LIN {X 0,Y 412.001,Z 515.214,A -85,B 0,C 180,E1 20178.098,E2 20178.098} C_VEL
LIN {X 0,Y 410.849,Z 527.535,A -85,B 0,C 180,E1 20175.962,E2 20175.962} C_VEL
LIN {X 0,Y 409.965,Z 537.694,A -85,B 0,C 180,E1 20173.828,E2 20173.828} C_VEL
LIN {X 0,Y 409.279,Z 546.504,A -85,B 0,C 180,E1 20171.556,E2 20171.556} C_VEL
LIN {X 0,Y 408.795,Z 553.889,A -85,B 0,C 180,E1 20169.148,E2 20169.148} C_VEL
LIN {X 0,Y 408.509,Z 559.483,A -85,B 0,C 180,E1 20166.747,E2 20166.747} C_VEL
LIN {X 0,Y 408.352,Z 563.605,A -85,B 0,C 180,E1 20164.213,E2 20164.213} C_VEL
LIN {X 0,Y 408.3,Z 565.991,A -85,B 0,C 180,E1 20161.684,E2 20161.684} C_VEL
LIN {X 0,Y 408.33,Z 566.694,A -85,B 0,C 180,E1 20159.158,E2 20159.158} C_VEL
LIN {X 0,Y 408.415,Z 565.71,A -85,B 0,C 180,E1 20156.632,E2 20156.632} C_VEL
LIN {X 0,Y 408.601,Z 563.017,A -85,B 0,C 180,E1 20154.101,E2 20154.101} C_VEL
LIN {X 0,Y 408.959,Z 558.554,A -85,B 0,C 180,E1 20151.565,E2 20151.565} C_VEL
LIN {X 0,Y 409.485,Z 552.563,A -85,B 0,C 180,E1 20149.163,E2 20149.163} C_VEL
LIN {X 0,Y 410.267,Z 544.675,A -85,B 0,C 180,E1 20146.757,E2 20146.757} C_VEL
LIN {X 0,Y 411.283,Z 535.28,A -85,B 0,C 180,E1 20144.49,E2 20144.49} C_VEL
LIN {X 0,Y 412.49,Z 524.341,A -85,B 0,C 180,E1 20142.363,E2 20142.363} C_VEL
LIN {X 0,Y 413.923,Z 511.401,A -85,B 0,C 180,E1 20140.308,E2 20140.308} C_VEL
LIN {X 0,Y 415.368,Z 497.854,A -85,B 0,C 180,E1 20138.538,E2 20138.538} C_VEL
LIN {X 0,Y 416.946,Z 482.078,A -85,B 0,C 180,E1 20136.842,E2 20136.842} C_VEL
LIN {X 0,Y 418.392,Z 465.945,A -85,B 0,C 180,E1 20135.429,E2 20135.429} C_VEL
LIN {X 0,Y 419.811,Z 447.969,A -85,B 0,C 180,E1 20134.161,E2 20134.161} C_VEL
LIN {X 0,Y 420.947,Z 429.995,A -85,B 0,C 180,E1 20133.173,E2 20133.173} C_VEL
LIN {X 0,Y 421.921,Z 409.848,A -85,B 0,C 180,E1 20132.352,E2 20132.352} C_VEL
LIN {X 0,Y 422.702,Z 387.891,A -85,B 0,C 180,E1 20131.742,E2 20131.742} C_VEL
LIN {X 0,Y 426.509,Z 310.931,A -85,B 0,C 180,E1 20129.855,E2 20129.855} C_VEL
LIN {X 0,Y 432.615,Z 224.265,A -85,B 0,C 180,E1 20127.543,E2 20127.543} C_VEL
LIN {X 0,Y 433.99,Z 205.725,A -85,B 0,C 180,E1 20127.01,E2 20127.01} C_VEL
LIN {X 0,Y 433.256,Z 198.82,A -85,B 0,C 180,E1 20126.606,E2 20126.606} C_VEL
LIN {X 0,Y 435.606,Z 168.281,A -85,B 0,C 180,E1 20123.85,E2 20123.85} C_VEL
LIN {X 0,Y 433.108,Z 159.078,A -85,B 0,C 180,E1 20122.283,E2 20122.283} C_VEL
LIN {X 0,Y 431.039,Z 153.151,A -85,B 0,C 180,E1 20120.995,E2 20120.995} C_VEL
LIN {X 0,Y 428.796,Z 147.265,A -85,B 0,C 180,E1 20119.416,E2 20119.416} C_VEL
LIN {X 0,Y 427.075,Z 143.317,A -85,B 0,C 180,E1 20117.916,E2 20117.916} C_VEL
LIN {X 0,Y 425.454,Z 140.615,A -85,B 0,C 180,E1 20115.735,E2 20115.735} C_VEL
LIN {X 0,Y 425.373,Z 139.927,A -85,B 0,C 180,E1 20114.891,E2 20114.891} C_VEL
LIN {X 0,Y 423.798,Z 146.299,A -85,B 0,C 180,E1 20113.08,E2 20113.08} C_VEL
LIN {X 0,Y 423.759,Z 151.293,A -85,B 0,C 180,E1 20111.84,E2 20111.84} C_VEL
LIN {X 0,Y 429.231,Z 165.38,A -85,B 0,C 180,E1 20109.893,E2 20109.893} C_VEL
LIN {X 0,Y 433.001,Z 172.844,A -85,B 0,C 180,E1 20109.358,E2 20109.358} C_VEL
LIN {X 0,Y 435.532,Z 195.035,A -85,B 0,C 180,E1 20108.647,E2 20108.647} C_VEL
LIN {X 0,Y 429.296,Z 412.636,A -85,B 0,C 180,E1 20104.609,E2 20104.609} C_VEL
LIN {X 0,Y 428.191,Z 433.533,A -85,B 0,C 180,E1 20104.074,E2 20104.074} C_VEL
LIN {X 0,Y 426.623,Z 453.74,A -85,B 0,C 180,E1 20103.327,E2 20103.327} C_VEL
LIN {X 0,Y 424.705,Z 474.23,A -85,B 0,C 180,E1 20102.305,E2 20102.305} C_VEL
LIN {X 0,Y 422.546,Z 493.789,A -85,B 0,C 180,E1 20101.055,E2 20101.055} C_VEL
LIN {X 0,Y 420.285,Z 512.438,A -85,B 0,C 180,E1 20099.581,E2 20099.581} C_VEL
LIN {X 0,Y 418.096,Z 529.523,A -85,B 0,C 180,E1 20097.952,E2 20097.952} C_VEL
LIN {X 0,Y 415.867,Z 546.483,A -85,B 0,C 180,E1 20096.027,E2 20096.027} C_VEL
LIN {X 0,Y 413.81,Z 562.406,A -85,B 0,C 180,E1 20093.874,E2 20093.874} C_VEL
LIN {X 0,Y 412.081,Z 576.353,A -85,B 0,C 180,E1 20091.643,E2 20091.643} C_VEL
LIN {X 0,Y 410.629,Z 589.282,A -85,B 0,C 180,E1 20089.192,E2 20089.192} C_VEL
LIN {X 0,Y 409.52,Z 600.704,A -85,B 0,C 180,E1 20086.599,E2 20086.599} C_VEL
LIN {X 0,Y 408.748,Z 610.548,A -85,B 0,C 180,E1 20083.871,E2 20083.871} C_VEL
LIN {X 0,Y 408.316,Z 618.348,A -85,B 0,C 180,E1 20081.155,E2 20081.155} C_VEL
LIN {X 0,Y 408.116,Z 624.334,A -85,B 0,C 180,E1 20078.454,E2 20078.454} C_VEL
LIN {X 0,Y 408.063,Z 628.633,A -85,B 0,C 180,E1 20075.767,E2 20075.767} C_VEL
LIN {X 0,Y 408.071,Z 631.328,A -85,B 0,C 180,E1 20073.091,E2 20073.091} C_VEL
LIN {X 0,Y 408.085,Z 632.331,A -85,B 0,C 180,E1 20070.422,E2 20070.422} C_VEL
LIN {X 0,Y 408.075,Z 631.775,A -85,B 0,C 180,E1 20067.754,E2 20067.754} C_VEL
LIN {X 0,Y 408.06,Z 629.669,A -85,B 0,C 180,E1 20065.081,E2 20065.081} C_VEL
LIN {X 0,Y 408.086,Z 625.91,A -85,B 0,C 180,E1 20062.398,E2 20062.398} C_VEL
LIN {X 0,Y 408.22,Z 620.753,A -85,B 0,C 180,E1 20059.844,E2 20059.844} C_VEL
LIN {X 0,Y 408.554,Z 613.61,A -85,B 0,C 180,E1 20057.133,E2 20057.133} C_VEL
LIN {X 0,Y 409.151,Z 605.098,A -85,B 0,C 180,E1 20054.553,E2 20054.553} C_VEL
LIN {X 0,Y 410.081,Z 594.653,A -85,B 0,C 180,E1 20051.963,E2 20051.963} C_VEL
LIN {X 0,Y 411.428,Z 581.988,A -85,B 0,C 180,E1 20049.368,E2 20049.368} C_VEL
LIN {X 0,Y 413.037,Z 568.55,A -85,B 0,C 180,E1 20047.063,E2 20047.063} C_VEL
LIN {X 0,Y 414.922,Z 553.715,A -85,B 0,C 180,E1 20044.906,E2 20044.906} C_VEL
LIN {X 0,Y 417.057,Z 537.409,A -85,B 0,C 180,E1 20042.903,E2 20042.903} C_VEL
LIN {X 0,Y 419.4,Z 519.234,A -85,B 0,C 180,E1 20041.037,E2 20041.037} C_VEL
LIN {X 0,Y 421.766,Z 500.31,A -85,B 0,C 180,E1 20039.437,E2 20039.437} C_VEL
LIN {X 0,Y 423.939,Z 481.065,A -85,B 0,C 180,E1 20038.109,E2 20038.109} C_VEL
LIN {X 0,Y 425.899,Z 461.768,A -85,B 0,C 180,E1 20037.047,E2 20037.047} C_VEL
LIN {X 0,Y 427.63,Z 441.297,A -85,B 0,C 180,E1 20036.184,E2 20036.184} C_VEL
LIN {X 0,Y 429.023,Z 419.453,A -85,B 0,C 180,E1 20035.539,E2 20035.539} C_VEL
LIN {X 0,Y 434.819,Z 218.607,A -85,B 0,C 180,E1 20031.785,E2 20031.785} C_VEL
LIN {X 0,Y 435.397,Z 192.267,A -85,B 0,C 180,E1 20031.286,E2 20031.286} C_VEL
LIN {X 0,Y 432.688,Z 171.767,A -85,B 0,C 180,E1 20030.595,E2 20030.595} C_VEL
LIN {X 0,Y 428.726,Z 164.272,A -85,B 0,C 180,E1 20030.006,E2 20030.006} C_VEL
LIN {X 0,Y 421.635,Z 146.282,A -85,B 0,C 180,E1 20027.418,E2 20027.418} C_VEL
LIN {X 0,Y 414.514,Z 130.026,A -85,B 0,C 180,E1 20024.835,E2 20024.835} C_VEL
LIN {X 0,Y 410.976,Z 122.341,A -85,B 0,C 180,E1 20023.512,E2 20023.512} C_VEL
LIN {X 0,Y 409.495,Z 119.111,A -85,B 0,C 180,E1 20022.94,E2 20022.94} C_VEL
LIN {X 0,Y 409.394,Z 118.478,A -85,B 0,C 180,E1 20022.802,E2 20022.802} C_VEL
LIN {X 0,Y 409.381,Z 118.43,A -85,B 0,C 180,E1 20019.045,E2 20019.045} C_VEL
LIN {X 0,Y 409.389,Z 118.489,A -85,B 0,C 180,E1 20015.099,E2 20015.099} C_VEL
LIN {X 0,Y 409.387,Z 118.49,A -85,B 0,C 180,E1 20011.183,E2 20011.183} C_VEL
LIN {X 0,Y 409.385,Z 118.487,A -85,B 0,C 180,E1 20007.253,E2 20007.253} C_VEL
LIN {X 0,Y 409.384,Z 118.474,A -85,B 0,C 180,E1 20003.307,E2 20003.307} C_VEL
LIN {X 0,Y 409.383,Z 118.471,A -85,B 0,C 180,E1 19999.4,E2 19999.4} C_VEL
LIN {X 0,Y 409.382,Z 118.488,A -85,B 0,C 180,E1 19995.439,E2 19995.439} C_VEL
LIN {X 0,Y 409.383,Z 118.482,A -85,B 0,C 180,E1 19991.553,E2 19991.553} C_VEL
LIN {X 0,Y 409.384,Z 118.465,A -85,B 0,C 180,E1 19987.72,E2 19987.72} C_VEL
LIN {X 0,Y 409.395,Z 118.489,A -85,B 0,C 180,E1 19983.921,E2 19983.921} C_VEL
LIN {X 0,Y 409.405,Z 118.465,A -85,B 0,C 180,E1 19980.14,E2 19980.14} C_VEL
LIN {X 0,Y 409.416,Z 118.476,A -85,B 0,C 180,E1 19976.359,E2 19976.359} C_VEL
LIN {X 0,Y 409.427,Z 118.48,A -85,B 0,C 180,E1 19972.422,E2 19972.422} C_VEL
LIN {X 0,Y 409.416,Z 118.461,A -85,B 0,C 180,E1 19968.448,E2 19968.448} C_VEL
LIN {X 0,Y 409.426,Z 118.482,A -85,B 0,C 180,E1 19964.562,E2 19964.562} C_VEL
LIN {X 0,Y 409.417,Z 118.478,A -85,B 0,C 180,E1 19960.601,E2 19960.601} C_VEL
LIN {X 0,Y 409.417,Z 118.463,A -85,B 0,C 180,E1 19956.668,E2 19956.668} C_VEL
LIN {X 0,Y 409.417,Z 118.47,A -85,B 0,C 180,E1 19952.669,E2 19952.669} C_VEL
LIN {X 0,Y 409.419,Z 118.484,A -85,B 0,C 180,E1 19948.73,E2 19948.73} C_VEL
LIN {X 0,Y 409.409,Z 118.488,A -85,B 0,C 180,E1 19944.805,E2 19944.805} C_VEL
LIN {X 0,Y 409.423,Z 118.489,A -85,B 0,C 180,E1 19940.764,E2 19940.764} C_VEL
LIN {X 0,Y 409.407,Z 118.486,A -85,B 0,C 180,E1 19936.857,E2 19936.857} C_VEL
LIN {X 0,Y 409.429,Z 118.668,A -85,B 0,C 180,E1 19932.947,E2 19932.947} C_VEL
LIN {X 0,Y 416.973,Z 136.874,A -85,B 0,C 180,E1 19929.573,E2 19929.573} C_VEL
LIN {X 0,Y 423.523,Z 154.25,A -85,B 0,C 180,E1 19926.674,E2 19926.674} C_VEL
LIN {X 0,Y 428.061,Z 168.125,A -85,B 0,C 180,E1 19924.581,E2 19924.581} C_VEL
LIN {X 0,Y 427.595,Z 173.606,A -85,B 0,C 180,E1 19924.047,E2 19924.047} C_VEL
LIN {X 0,Y 433.281,Z 207.319,A -85,B 0,C 180,E1 19922.841,E2 19922.841} C_VEL
LIN {X 0,Y 429.712,Z 391.959,A -85,B 0,C 180,E1 19919.803,E2 19919.803} C_VEL
LIN {X 0,Y 428.766,Z 411.13,A -85,B 0,C 180,E1 19919.244,E2 19919.244} C_VEL
LIN {X 0,Y 427.491,Z 428.701,A -85,B 0,C 180,E1 19918.497,E2 19918.497} C_VEL
LIN {X 0,Y 425.737,Z 446.594,A -85,B 0,C 180,E1 19917.482,E2 19917.482} C_VEL
LIN {X 0,Y 424.972,Z 453.23,A -85,B 0,C 180,E1 19917.028,E2 19917.028} C_VEL
LIN {X 0,Y 423.297,Z 460.11,A -85,B 0,C 180,E1 19916.595,E2 19916.595} C_VEL
LIN {X 0,Y 416.045,Z 476.098,A -85,B 0,C 180,E1 19915.6,E2 19915.6} C_VEL
LIN {X 0,Y 413.969,Z 482.401,A -85,B 0,C 180,E1 19915.045,E2 19915.045} C_VEL
LIN {X 0,Y 413.808,Z 483.266,A -85,B 0,C 180,E1 19914.953,E2 19914.953} C_VEL
LIN {X 0,Y 411.333,Z 498.226,A -85,B 0,C 180,E1 19913.189,E2 19913.189} C_VEL
LIN {X 0,Y 408.923,Z 511.954,A -85,B 0,C 180,E1 19911.214,E2 19911.214} C_VEL
LIN {X 0,Y 406.723,Z 524.135,A -85,B 0,C 180,E1 19909.083,E2 19909.083} C_VEL
LIN {X 0,Y 404.695,Z 535.458,A -85,B 0,C 180,E1 19906.653,E2 19906.653} C_VEL
LIN {X 0,Y 403.144,Z 544.622,A -85,B 0,C 180,E1 19904.212,E2 19904.212} C_VEL
LIN {X 0,Y 401.948,Z 552.334,A -85,B 0,C 180,E1 19901.623,E2 19901.623} C_VEL
LIN {X 0,Y 401.123,Z 558.537,A -85,B 0,C 180,E1 19898.889,E2 19898.889} C_VEL
LIN {X 0,Y 400.638,Z 562.943,A -85,B 0,C 180,E1 19896.16,E2 19896.16} C_VEL
LIN {X 0,Y 400.393,Z 565.694,A -85,B 0,C 180,E1 19893.435,E2 19893.435} C_VEL
LIN {X 0,Y 400.312,Z 566.904,A -85,B 0,C 180,E1 19890.572,E2 19890.572} C_VEL
LIN {X 0,Y 400.345,Z 566.429,A -85,B 0,C 180,E1 19887.709,E2 19887.709} C_VEL
LIN {X 0,Y 400.517,Z 564.249,A -85,B 0,C 180,E1 19884.843,E2 19884.843} C_VEL
LIN {X 0,Y 400.893,Z 560.519,A -85,B 0,C 180,E1 19882.115,E2 19882.115} C_VEL
LIN {X 0,Y 401.567,Z 555.06,A -85,B 0,C 180,E1 19879.382,E2 19879.382} C_VEL
LIN {X 0,Y 402.583,Z 548.135,A -85,B 0,C 180,E1 19876.791,E2 19876.791} C_VEL
LIN {X 0,Y 403.961,Z 539.762,A -85,B 0,C 180,E1 19874.33,E2 19874.33} C_VEL
LIN {X 0,Y 405.763,Z 529.521,A -85,B 0,C 180,E1 19871.911,E2 19871.911} C_VEL
LIN {X 0,Y 407.773,Z 518.446,A -85,B 0,C 180,E1 19869.773,E2 19869.773} C_VEL
LIN {X 0,Y 410.162,Z 505.064,A -85,B 0,C 180,E1 19867.648,E2 19867.648} C_VEL
LIN {X 0,Y 412.569,Z 491.037,A -85,B 0,C 180,E1 19865.821,E2 19865.821} C_VEL
LIN {X 0,Y 414.94,Z 476.063,A -85,B 0,C 180,E1 19864.218,E2 19864.218} C_VEL
LIN {X 0,Y 417.282,Z 459.337,A -85,B 0,C 180,E1 19862.763,E2 19862.763} C_VEL
LIN {X 0,Y 419.315,Z 442.433,A -85,B 0,C 180,E1 19861.594,E2 19861.594} C_VEL
LIN {X 0,Y 421.075,Z 423.922,A -85,B 0,C 180,E1 19860.605,E2 19860.605} C_VEL
LIN {X 0,Y 422.376,Z 405.228,A -85,B 0,C 180,E1 19859.881,E2 19859.881} C_VEL
LIN {X 0,Y 423.174,Z 385.891,A -85,B 0,C 180,E1 19859.393,E2 19859.393} C_VEL
LIN {X 0,Y 426.735,Z 207.213,A -85,B 0,C 180,E1 19856.418,E2 19856.418} C_VEL
LIN {X 0,Y 420.91,Z 172.733,A -85,B 0,C 180,E1 19855.117,E2 19855.117} C_VEL
LIN {X 0,Y 420.855,Z 170.187,A -85,B 0,C 180,E1 19854.813,E2 19854.813} C_VEL
LIN {X 0,Y 414.806,Z 152.486,A -85,B 0,C 180,E1 19852.019,E2 19852.019} C_VEL
LIN {X 0,Y 408.812,Z 137.026,A -85,B 0,C 180,E1 19849.305,E2 19849.305} C_VEL
LIN {X 0,Y 402.949,Z 123.185,A -85,B 0,C 180,E1 19846.639,E2 19846.639} C_VEL
LIN {X 0,Y 401.542,Z 119.781,A -85,B 0,C 180,E1 19845.958,E2 19845.958} C_VEL
LIN {X 0,Y 401.501,Z 119.467,A -85,B 0,C 180,E1 19845.79,E2 19845.79} C_VEL
LIN {X 0,Y 401.504,Z 119.474,A -85,B 0,C 180,E1 19841.867,E2 19841.867} C_VEL
LIN {X 0,Y 401.535,Z 119.694,A -85,B 0,C 180,E1 19840.14,E2 19840.14} C_VEL
LIN {X 0,Y 411.347,Z 145.789,A -85,B 0,C 180,E1 19836.724,E2 19836.724} C_VEL
LIN {X 0,Y 417.493,Z 164.195,A -85,B 0,C 180,E1 19834.46,E2 19834.46} C_VEL
LIN {X 0,Y 416.544,Z 185.557,A -85,B 0,C 180,E1 19832.581,E2 19832.581} C_VEL
LIN {X 0,Y 419.192,Z 205.833,A -85,B 0,C 180,E1 19831.896,E2 19831.896} C_VEL
LIN {X 0,Y 413.156,Z 396.893,A -85,B 0,C 180,E1 19827.859,E2 19827.859} C_VEL
LIN {X 0,Y 412.314,Z 416.605,A -85,B 0,C 180,E1 19827.172,E2 19827.172} C_VEL
LIN {X 0,Y 411.233,Z 435.212,A -85,B 0,C 180,E1 19826.264,E2 19826.264} C_VEL
LIN {X 0,Y 409.928,Z 453.331,A -85,B 0,C 180,E1 19825.113,E2 19825.113} C_VEL
LIN {X 0,Y 408.44,Z 471.321,A -85,B 0,C 180,E1 19823.671,E2 19823.671} C_VEL
LIN {X 0,Y 406.971,Z 487.399,A -85,B 0,C 180,E1 19822.08,E2 19822.08} C_VEL
LIN {X 0,Y 405.512,Z 502.478,A -85,B 0,C 180,E1 19820.269,E2 19820.269} C_VEL
LIN {X 0,Y 404.18,Z 515.942,A -85,B 0,C 180,E1 19818.311,E2 19818.311} C_VEL
LIN {X 0,Y 402.977,Z 528.27,A -85,B 0,C 180,E1 19816.135,E2 19816.135} C_VEL
LIN {X 0,Y 402.054,Z 538.437,A -85,B 0,C 180,E1 19813.959,E2 19813.959} C_VEL
LIN {X 0,Y 401.338,Z 547.254,A -85,B 0,C 180,E1 19811.642,E2 19811.642} C_VEL
LIN {X 0,Y 400.832,Z 554.643,A -85,B 0,C 180,E1 19809.187,E2 19809.187} C_VEL
LIN {X 0,Y 400.536,Z 560.236,A -85,B 0,C 180,E1 19806.738,E2 19806.738} C_VEL
LIN {X 0,Y 400.377,Z 564.352,A -85,B 0,C 180,E1 19804.153,E2 19804.153} C_VEL
LIN {X 0,Y 400.327,Z 566.721,A -85,B 0,C 180,E1 19801.575,E2 19801.575} C_VEL
LIN {X 0,Y 400.361,Z 567.391,A -85,B 0,C 180,E1 19798.999,E2 19798.999} C_VEL
LIN {X 0,Y 400.469,Z 566.369,A -85,B 0,C 180,E1 19796.422,E2 19796.422} C_VEL
LIN {X 0,Y 400.685,Z 563.635,A -85,B 0,C 180,E1 19793.841,E2 19793.841} C_VEL
LIN {X 0,Y 401.059,Z 559.39,A -85,B 0,C 180,E1 19791.398,E2 19791.398} C_VEL
LIN {X 0,Y 401.641,Z 553.441,A -85,B 0,C 180,E1 19788.949,E2 19788.949} C_VEL
LIN {X 0,Y 402.433,Z 546.106,A -85,B 0,C 180,E1 19786.641,E2 19786.641} C_VEL
LIN {X 0,Y 403.507,Z 536.829,A -85,B 0,C 180,E1 19784.33,E2 19784.33} C_VEL
LIN {X 0,Y 404.802,Z 526.128,A -85,B 0,C 180,E1 19782.165,E2 19782.165} C_VEL
LIN {X 0,Y 406.267,Z 513.905,A -85,B 0,C 180,E1 19780.146,E2 19780.146} C_VEL
LIN {X 0,Y 407.928,Z 499.555,A -85,B 0,C 180,E1 19778.202,E2 19778.202} C_VEL
LIN {X 0,Y 409.528,Z 484.657,A -85,B 0,C 180,E1 19776.549,E2 19776.549} C_VEL
LIN {X 0,Y 411.149,Z 468.135,A -85,B 0,C 180,E1 19775.044,E2 19775.044} C_VEL
LIN {X 0,Y 412.649,Z 450.503,A -85,B 0,C 180,E1 19773.756,E2 19773.756} C_VEL
LIN {X 0,Y 413.977,Z 431.928,A -85,B 0,C 180,E1 19772.684,E2 19772.684} C_VEL
LIN {X 0,Y 415.037,Z 412.33,A -85,B 0,C 180,E1 19771.848,E2 19771.848} C_VEL
LIN {X 0,Y 415.957,Z 389.581,A -85,B 0,C 180,E1 19771.177,E2 19771.177} C_VEL
LIN {X 0,Y 419.985,Z 316.38,A -85,B 0,C 180,E1 19769.307,E2 19769.307} C_VEL
LIN {X 0,Y 426.604,Z 230.848,A -85,B 0,C 180,E1 19766.941,E2 19766.941} C_VEL
LIN {X 0,Y 428.6,Z 207.571,A -85,B 0,C 180,E1 19766.252,E2 19766.252} C_VEL
LIN {X 0,Y 427.98,Z 199.565,A -85,B 0,C 180,E1 19765.735,E2 19765.735} C_VEL
LIN {X 0,Y 430.469,Z 172.638,A -85,B 0,C 180,E1 19763.259,E2 19763.259} C_VEL
LIN {X 0,Y 428.535,Z 164.639,A -85,B 0,C 180,E1 19761.808,E2 19761.808} C_VEL
LIN {X 0,Y 426.436,Z 158.021,A -85,B 0,C 180,E1 19760.27,E2 19760.27} C_VEL
LIN {X 0,Y 424.798,Z 153.51,A -85,B 0,C 180,E1 19758.869,E2 19758.869} C_VEL
LIN {X 0,Y 423.624,Z 150.051,A -85,B 0,C 180,E1 19757.426,E2 19757.426} C_VEL
LIN {X 0,Y 422.617,Z 147.609,A -85,B 0,C 180,E1 19755.216,E2 19755.216} C_VEL
LIN {X 0,Y 422.516,Z 147.909,A -85,B 0,C 180,E1 19754.963,E2 19754.963} C_VEL
LIN {X 0,Y 421.078,Z 153.176,A -85,B 0,C 180,E1 19753.521,E2 19753.521} C_VEL
LIN {X 0,Y 420.701,Z 159.091,A -85,B 0,C 180,E1 19752.085,E2 19752.085} C_VEL
LIN {X 0,Y 421.413,Z 165.842,A -85,B 0,C 180,E1 19750.689,E2 19750.689} C_VEL
LIN {X 0,Y 426.814,Z 176.179,A -85,B 0,C 180,E1 19749.903,E2 19749.903} C_VEL
LIN {X 0,Y 429.026,Z 196.097,A -85,B 0,C 180,E1 19749.253,E2 19749.253} C_VEL
LIN {X 0,Y 422.506,Z 412.542,A -85,B 0,C 180,E1 19745.182,E2 19745.182} C_VEL
LIN {X 0,Y 421.342,Z 433.504,A -85,B 0,C 180,E1 19744.635,E2 19744.635} C_VEL
LIN {X 0,Y 419.701,Z 453.581,A -85,B 0,C 180,E1 19743.881,E2 19743.881} C_VEL
LIN {X 0,Y 417.728,Z 473.639,A -85,B 0,C 180,E1 19742.868,E2 19742.868} C_VEL
LIN {X 0,Y 415.391,Z 493.795,A -85,B 0,C 180,E1 19741.561,E2 19741.561} C_VEL
LIN {X 0,Y 412.918,Z 513.085,A -85,B 0,C 180,E1 19740.003,E2 19740.003} C_VEL
LIN {X 0,Y 410.527,Z 530.653,A -85,B 0,C 180,E1 19738.277,E2 19738.277} C_VEL
LIN {X 0,Y 408.195,Z 547.333,A -85,B 0,C 180,E1 19736.319,E2 19736.319} C_VEL
LIN {X 0,Y 406.105,Z 562.533,A -85,B 0,C 180,E1 19734.202,E2 19734.202} C_VEL
LIN {X 0,Y 404.179,Z 577.17,A -85,B 0,C 180,E1 19731.782,E2 19731.782} C_VEL
LIN {X 0,Y 402.673,Z 589.852,A -85,B 0,C 180,E1 19729.285,E2 19729.285} C_VEL
LIN {X 0,Y 401.581,Z 600.503,A -85,B 0,C 180,E1 19726.788,E2 19726.788} C_VEL
LIN {X 0,Y 400.775,Z 610.275,A -85,B 0,C 180,E1 19724.005,E2 19724.005} C_VEL
LIN {X 0,Y 400.325,Z 618.019,A -85,B 0,C 180,E1 19721.235,E2 19721.235} C_VEL
LIN {X 0,Y 400.125,Z 623.925,A -85,B 0,C 180,E1 19718.479,E2 19718.479} C_VEL
LIN {X 0,Y 400.08,Z 628.143,A -85,B 0,C 180,E1 19715.738,E2 19715.738} C_VEL
LIN {X 0,Y 400.096,Z 630.754,A -85,B 0,C 180,E1 19713.009,E2 19713.009} C_VEL
LIN {X 0,Y 400.115,Z 631.71,A -85,B 0,C 180,E1 19710.287,E2 19710.287} C_VEL
LIN {X 0,Y 400.099,Z 631.052,A -85,B 0,C 180,E1 19707.566,E2 19707.566} C_VEL
LIN {X 0,Y 400.079,Z 628.835,A -85,B 0,C 180,E1 19704.839,E2 19704.839} C_VEL
LIN {X 0,Y 400.11,Z 625.009,A -85,B 0,C 180,E1 19702.101,E2 19702.101} C_VEL
LIN {X 0,Y 400.269,Z 619.401,A -85,B 0,C 180,E1 19699.349,E2 19699.349} C_VEL
LIN {X 0,Y 400.649,Z 612.018,A -85,B 0,C 180,E1 19696.581,E2 19696.581} C_VEL
LIN {X 0,Y 401.376,Z 602.701,A -85,B 0,C 180,E1 19693.8,E2 19693.8} C_VEL
LIN {X 0,Y 402.448,Z 591.876,A -85,B 0,C 180,E1 19691.158,E2 19691.158} C_VEL
LIN {X 0,Y 403.88,Z 579.609,A -85,B 0,C 180,E1 19688.66,E2 19688.66} C_VEL
LIN {X 0,Y 405.656,Z 565.925,A -85,B 0,C 180,E1 19686.313,E2 19686.313} C_VEL
LIN {X 0,Y 407.803,Z 550.192,A -85,B 0,C 180,E1 19684.047,E2 19684.047} C_VEL
LIN {X 0,Y 410.164,Z 533.328,A -85,B 0,C 180,E1 19682.015,E2 19682.015} C_VEL
LIN {X 0,Y 412.584,Z 515.406,A -85,B 0,C 180,E1 19680.213,E2 19680.213} C_VEL
LIN {X 0,Y 414.918,Z 497.379,A -85,B 0,C 180,E1 19678.716,E2 19678.716} C_VEL
LIN {X 0,Y 417.122,Z 478.715,A -85,B 0,C 180,E1 19677.444,E2 19677.444} C_VEL
LIN {X 0,Y 419.259,Z 458.139,A -85,B 0,C 180,E1 19676.336,E2 19676.336} C_VEL
LIN {X 0,Y 421.003,Z 437.587,A -85,B 0,C 180,E1 19675.502,E2 19675.502} C_VEL
LIN {X 0,Y 422.324,Z 416.696,A -85,B 0,C 180,E1 19674.911,E2 19674.911} C_VEL
LIN {X 0,Y 428.603,Z 209.098,A -85,B 0,C 180,E1 19670.989,E2 19670.989} C_VEL
LIN {X 0,Y 428.877,Z 193.319,A -85,B 0,C 180,E1 19670.678,E2 19670.678} C_VEL
LIN {X 0,Y 426.492,Z 175.187,A -85,B 0,C 180,E1 19670.05,E2 19670.05} C_VEL
LIN {X 0,Y 420.756,Z 164.509,A -85,B 0,C 180,E1 19669.196,E2 19669.196} C_VEL
LIN {X 0,Y 413.184,Z 145.601,A -85,B 0,C 180,E1 19666.348,E2 19666.348} C_VEL
LIN {X 0,Y 405.15,Z 127.665,A -85,B 0,C 180,E1 19663.319,E2 19663.319} C_VEL
LIN {X 0,Y 401.761,Z 120.757,A -85,B 0,C 180,E1 19662.025,E2 19662.025} C_VEL
LIN {X 0,Y 401.475,Z 119.477,A -85,B 0,C 180,E1 19661.784,E2 19661.784} C_VEL
LIN {X 0,Y 401.479,Z 119.412,A -85,B 0,C 180,E1 19657.962,E2 19657.962} C_VEL
LIN {X 0,Y 401.484,Z 119.465,A -85,B 0,C 180,E1 19653.975,E2 19653.975} C_VEL
LIN {X 0,Y 401.487,Z 119.468,A -85,B 0,C 180,E1 19650.037,E2 19650.037} C_VEL
LIN {X 0,Y 401.487,Z 119.475,A -85,B 0,C 180,E1 19646.155,E2 19646.155} C_VEL
LIN {X 0,Y 401.489,Z 119.47,A -85,B 0,C 180,E1 19642.12,E2 19642.12} C_VEL
LIN {X 0,Y 401.479,Z 119.454,A -85,B 0,C 180,E1 19638.138,E2 19638.138} C_VEL
LIN {X 0,Y 401.493,Z 119.455,A -85,B 0,C 180,E1 19634.273,E2 19634.273} C_VEL
LIN {X 0,Y 401.484,Z 119.476,A -85,B 0,C 180,E1 19630.329,E2 19630.329} C_VEL
LIN {X 0,Y 401.488,Z 119.448,A -85,B 0,C 180,E1 19626.434,E2 19626.434} C_VEL
LIN {X 0,Y 401.48,Z 119.46,A -85,B 0,C 180,E1 19622.426,E2 19622.426} C_VEL
LIN {X 0,Y 401.48,Z 119.47,A -85,B 0,C 180,E1 19618.573,E2 19618.573} C_VEL
LIN {X 0,Y 401.477,Z 119.448,A -85,B 0,C 180,E1 19614.569,E2 19614.569} C_VEL
LIN {X 0,Y 401.473,Z 119.474,A -85,B 0,C 180,E1 19610.684,E2 19610.684} C_VEL
LIN {X 0,Y 401.471,Z 119.464,A -85,B 0,C 180,E1 19606.754,E2 19606.754} C_VEL
LIN {X 0,Y 401.456,Z 119.455,A -85,B 0,C 180,E1 19602.909,E2 19602.909} C_VEL
LIN {X 0,Y 401.457,Z 119.478,A -85,B 0,C 180,E1 19598.983,E2 19598.983} C_VEL
LIN {X 0,Y 401.447,Z 119.47,A -85,B 0,C 180,E1 19595.107,E2 19595.107} C_VEL
LIN {X 0,Y 401.442,Z 119.455,A -85,B 0,C 180,E1 19591.246,E2 19591.246} C_VEL
LIN {X 0,Y 401.434,Z 119.464,A -85,B 0,C 180,E1 19587.452,E2 19587.452} C_VEL
LIN {X 0,Y 401.431,Z 119.472,A -85,B 0,C 180,E1 19583.561,E2 19583.561} C_VEL
LIN {X 0,Y 401.429,Z 119.472,A -85,B 0,C 180,E1 19579.639,E2 19579.639} C_VEL
LIN {X 0,Y 401.428,Z 119.469,A -85,B 0,C 180,E1 19575.78,E2 19575.78} C_VEL
LIN {X 0,Y 401.453,Z 119.627,A -85,B 0,C 180,E1 19573.963,E2 19573.963} C_VEL
LIN {X 0,Y 402.705,Z 122.894,A -85,B 0,C 180,E1 19573.324,E2 19573.324} C_VEL
LIN {X 0,Y 408.238,Z 135.837,A -85,B 0,C 180,E1 19570.816,E2 19570.816} C_VEL
LIN {X 0,Y 414.115,Z 150.717,A -85,B 0,C 180,E1 19568.176,E2 19568.176} C_VEL
LIN {X 0,Y 420.15,Z 168.072,A -85,B 0,C 180,E1 19565.405,E2 19565.405} C_VEL
LIN {X 0,Y 421.005,Z 171.496,A -85,B 0,C 180,E1 19564.914,E2 19564.914} C_VEL
LIN {X 0,Y 420.942,Z 173.721,A -85,B 0,C 180,E1 19564.729,E2 19564.729} C_VEL
LIN {X 0,Y 426.778,Z 208.456,A -85,B 0,C 180,E1 19563.45,E2 19563.45} C_VEL
LIN {X 0,Y 422.973,Z 392.261,A -85,B 0,C 180,E1 19560.381,E2 19560.381} C_VEL
LIN {X 0,Y 421.979,Z 411.446,A -85,B 0,C 180,E1 19559.815,E2 19559.815} C_VEL
LIN {X 0,Y 420.551,Z 429.933,A -85,B 0,C 180,E1 19559.012,E2 19559.012} C_VEL
LIN {X 0,Y 418.717,Z 447.641,A -85,B 0,C 180,E1 19557.983,E2 19557.983} C_VEL
LIN {X 0,Y 416.612,Z 464.361,A -85,B 0,C 180,E1 19556.742,E2 19556.742} C_VEL
LIN {X 0,Y 414.204,Z 480.814,A -85,B 0,C 180,E1 19555.217,E2 19555.217} C_VEL
LIN {X 0,Y 413.808,Z 483.266,A -85,B 0,C 180,E1 19554.953,E2 19554.953} C_VEL
LIN {X 0,Y 411.935,Z 489.421,A -85,B 0,C 180,E1 19554.342,E2 19554.342} C_VEL
LIN {X 0,Y 403.942,Z 504.398,A -85,B 0,C 180,E1 19552.83,E2 19552.83} C_VEL
LIN {X 0,Y 402.036,Z 509.819,A -85,B 0,C 180,E1 19552.092,E2 19552.092} C_VEL
LIN {X 0,Y 399.597,Z 522.65,A -85,B 0,C 180,E1 19549.894,E2 19549.894} C_VEL
LIN {X 0,Y 397.474,Z 533.775,A -85,B 0,C 180,E1 19547.562,E2 19547.562} C_VEL
LIN {X 0,Y 395.723,Z 543.366,A -85,B 0,C 180,E1 19545.084,E2 19545.084} C_VEL
LIN {X 0,Y 394.338,Z 551.489,A -85,B 0,C 180,E1 19542.445,E2 19542.445} C_VEL
LIN {X 0,Y 393.362,Z 558.07,A -85,B 0,C 180,E1 19539.657,E2 19539.657} C_VEL
LIN {X 0,Y 392.776,Z 562.833,A -85,B 0,C 180,E1 19536.871,E2 19536.871} C_VEL
LIN {X 0,Y 392.47,Z 565.925,A -85,B 0,C 180,E1 19534.09,E2 19534.09} C_VEL
LIN {X 0,Y 392.349,Z 567.447,A -85,B 0,C 180,E1 19531.313,E2 19531.313} C_VEL
LIN {X 0,Y 392.356,Z 567.387,A -85,B 0,C 180,E1 19528.393,E2 19528.393} C_VEL
LIN {X 0,Y 392.496,Z 565.634,A -85,B 0,C 180,E1 19525.47,E2 19525.47} C_VEL
LIN {X 0,Y 392.836,Z 562.354,A -85,B 0,C 180,E1 19522.688,E2 19522.688} C_VEL
LIN {X 0,Y 393.462,Z 557.371,A -85,B 0,C 180,E1 19519.901,E2 19519.901} C_VEL
LIN {X 0,Y 394.498,Z 550.532,A -85,B 0,C 180,E1 19517.112,E2 19517.112} C_VEL
LIN {X 0,Y 395.945,Z 542.14,A -85,B 0,C 180,E1 19514.473,E2 19514.473} C_VEL
LIN {X 0,Y 397.773,Z 532.226,A -85,B 0,C 180,E1 19511.989,E2 19511.989} C_VEL
LIN {X 0,Y 399.963,Z 520.793,A -85,B 0,C 180,E1 19509.666,E2 19509.666} C_VEL
LIN {X 0,Y 402.309,Z 508.427,A -85,B 0,C 180,E1 19507.599,E2 19507.599} C_VEL
LIN {X 0,Y 404.823,Z 494.639,A -85,B 0,C 180,E1 19505.698,E2 19505.698} C_VEL
LIN {X 0,Y 407.34,Z 479.794,A -85,B 0,C 180,E1 19504.013,E2 19504.013} C_VEL
LIN {X 0,Y 409.768,Z 463.824,A -85,B 0,C 180,E1 19502.536,E2 19502.536} C_VEL
LIN {X 0,Y 411.988,Z 446.876,A -85,B 0,C 180,E1 19501.279,E2 19501.279} C_VEL
LIN {X 0,Y 413.91,Z 428.784,A -85,B 0,C 180,E1 19500.236,E2 19500.236} C_VEL
LIN {X 0,Y 415.386,Z 409.956,A -85,B 0,C 180,E1 19499.434,E2 19499.434} C_VEL
LIN {X 0,Y 416.368,Z 390.878,A -85,B 0,C 180,E1 19498.887,E2 19498.887} C_VEL
LIN {X 0,Y 420.27,Z 208.498,A -85,B 0,C 180,E1 19495.79,E2 19495.79} C_VEL
LIN {X 0,Y 414.357,Z 174.162,A -85,B 0,C 180,E1 19494.469,E2 19494.469} C_VEL
LIN {X 0,Y 413.625,Z 172.49,A -85,B 0,C 180,E1 19494.313,E2 19494.313} C_VEL
LIN {X 0,Y 407.601,Z 154.876,A -85,B 0,C 180,E1 19491.458,E2 19491.458} C_VEL
LIN {X 0,Y 401.411,Z 138.902,A -85,B 0,C 180,E1 19488.569,E2 19488.569} C_VEL
LIN {X 0,Y 396.204,Z 127.109,A -85,B 0,C 180,E1 19486.199,E2 19486.199} C_VEL
LIN {X 0,Y 394.509,Z 123.355,A -85,B 0,C 180,E1 19485.408,E2 19485.408} C_VEL
LIN {X 0,Y 393.548,Z 120.463,A -85,B 0,C 180,E1 19484.816,E2 19484.816} C_VEL
LIN {X 0,Y 393.56,Z 120.5,A -85,B 0,C 180,E1 19480.831,E2 19480.831} C_VEL
LIN {X 0,Y 403.258,Z 146.151,A -85,B 0,C 180,E1 19477.407,E2 19477.407} C_VEL
LIN {X 0,Y 410.285,Z 166.847,A -85,B 0,C 180,E1 19474.811,E2 19474.811} C_VEL
LIN {X 0,Y 409.425,Z 186.05,A -85,B 0,C 180,E1 19473.115,E2 19473.115} C_VEL
LIN {X 0,Y 412.105,Z 206.928,A -85,B 0,C 180,E1 19472.397,E2 19472.397} C_VEL
LIN {X 0,Y 405.71,Z 397.5,A -85,B 0,C 180,E1 19468.261,E2 19468.261} C_VEL
LIN {X 0,Y 404.852,Z 416.768,A -85,B 0,C 180,E1 19467.578,E2 19467.578} C_VEL
LIN {X 0,Y 403.7,Z 435.787,A -85,B 0,C 180,E1 19466.634,E2 19466.634} C_VEL
LIN {X 0,Y 402.299,Z 454.447,A -85,B 0,C 180,E1 19465.423,E2 19465.423} C_VEL
LIN {X 0,Y 400.795,Z 471.924,A -85,B 0,C 180,E1 19463.994,E2 19463.994} C_VEL
LIN {X 0,Y 399.267,Z 488.032,A -85,B 0,C 180,E1 19462.374,E2 19462.374} C_VEL
LIN {X 0,Y 397.749,Z 503.148,A -85,B 0,C 180,E1 19460.529,E2 19460.529} C_VEL
LIN {X 0,Y 396.361,Z 516.632,A -85,B 0,C 180,E1 19458.533,E2 19458.533} C_VEL
LIN {X 0,Y 395.107,Z 528.991,A -85,B 0,C 180,E1 19456.314,E2 19456.314} C_VEL
LIN {X 0,Y 394.145,Z 539.176,A -85,B 0,C 180,E1 19454.095,E2 19454.095} C_VEL
LIN {X 0,Y 393.397,Z 548.004,A -85,B 0,C 180,E1 19451.732,E2 19451.732} C_VEL
LIN {X 0,Y 392.871,Z 555.399,A -85,B 0,C 180,E1 19449.227,E2 19449.227} C_VEL
LIN {X 0,Y 392.548,Z 561.261,A -85,B 0,C 180,E1 19446.582,E2 19446.582} C_VEL
LIN {X 0,Y 392.397,Z 565.268,A -85,B 0,C 180,E1 19443.945,E2 19443.945} C_VEL
LIN {X 0,Y 392.355,Z 567.529,A -85,B 0,C 180,E1 19441.315,E2 19441.315} C_VEL
LIN {X 0,Y 392.395,Z 568.095,A -85,B 0,C 180,E1 19438.832,E2 19438.832} C_VEL
LIN {X 0,Y 392.526,Z 567.04,A -85,B 0,C 180,E1 19436.203,E2 19436.203} C_VEL
LIN {X 0,Y 392.775,Z 564.259,A -85,B 0,C 180,E1 19433.569,E2 19433.569} C_VEL
LIN {X 0,Y 393.196,Z 559.98,A -85,B 0,C 180,E1 19431.077,E2 19431.077} C_VEL
LIN {X 0,Y 393.854,Z 553.962,A -85,B 0,C 180,E1 19428.579,E2 19428.579} C_VEL
LIN {X 0,Y 394.804,Z 546.046,A -85,B 0,C 180,E1 19426.079,E2 19426.079} C_VEL
LIN {X 0,Y 396.013,Z 536.584,A -85,B 0,C 180,E1 19423.725,E2 19423.725} C_VEL
LIN {X 0,Y 397.437,Z 525.563,A -85,B 0,C 180,E1 19421.52,E2 19421.52} C_VEL
LIN {X 0,Y 399.053,Z 513.069,A -85,B 0,C 180,E1 19419.465,E2 19419.465} C_VEL
LIN {X 0,Y 400.794,Z 498.95,A -85,B 0,C 180,E1 19417.562,E2 19417.562} C_VEL
LIN {X 0,Y 402.541,Z 483.864,A -85,B 0,C 180,E1 19415.884,E2 19415.884} C_VEL
LIN {X 0,Y 404.389,Z 466.151,A -85,B 0,C 180,E1 19414.283,E2 19414.283} C_VEL
LIN {X 0,Y 405.98,Z 448.387,A -85,B 0,C 180,E1 19413.01,E2 19413.01} C_VEL
LIN {X 0,Y 407.458,Z 428.274,A -85,B 0,C 180,E1 19411.891,E2 19411.891} C_VEL
LIN {X 0,Y 408.588,Z 408.522,A -85,B 0,C 180,E1 19411.079,E2 19411.079} C_VEL
LIN {X 0,Y 410.621,Z 367.602,A -85,B 0,C 180,E1 19409.964,E2 19409.964} C_VEL
LIN {X 0,Y 415.846,Z 292.509,A -85,B 0,C 180,E1 19407.897,E2 19407.897} C_VEL
LIN {X 0,Y 423.516,Z 210.155,A -85,B 0,C 180,E1 19405.497,E2 19405.497} C_VEL
LIN {X 0,Y 422.962,Z 201.048,A -85,B 0,C 180,E1 19404.879,E2 19404.879} C_VEL
LIN {X 0,Y 425.599,Z 177.145,A -85,B 0,C 180,E1 19402.637,E2 19402.637} C_VEL
LIN {X 0,Y 423.924,Z 169.3,A -85,B 0,C 180,E1 19401.109,E2 19401.109} C_VEL
LIN {X 0,Y 422.229,Z 163.269,A -85,B 0,C 180,E1 19399.546,E2 19399.546} C_VEL
LIN {X 0,Y 421.277,Z 160.309,A -85,B 0,C 180,E1 19398.534,E2 19398.534} C_VEL
LIN {X 0,Y 420.519,Z 157.356,A -85,B 0,C 180,E1 19397.283,E2 19397.283} C_VEL
LIN {X 0,Y 419.804,Z 155.382,A -85,B 0,C 180,E1 19395.264,E2 19395.264} C_VEL
LIN {X 0,Y 418.471,Z 159.845,A -85,B 0,C 180,E1 19394.013,E2 19394.013} C_VEL
LIN {X 0,Y 417.801,Z 165.395,A -85,B 0,C 180,E1 19392.631,E2 19392.631} C_VEL
LIN {X 0,Y 418.04,Z 172.246,A -85,B 0,C 180,E1 19391.22,E2 19391.22} C_VEL
LIN {X 0,Y 418.316,Z 174.871,A -85,B 0,C 180,E1 19390.818,E2 19390.818} C_VEL
LIN {X 0,Y 420.693,Z 179.75,A -85,B 0,C 180,E1 19390.457,E2 19390.457} C_VEL
LIN {X 0,Y 422.566,Z 197.305,A -85,B 0,C 180,E1 19389.876,E2 19389.876} C_VEL
LIN {X 0,Y 415.757,Z 412.585,A -85,B 0,C 180,E1 19385.772,E2 19385.772} C_VEL
LIN {X 0,Y 414.511,Z 433.782,A -85,B 0,C 180,E1 19385.206,E2 19385.206} C_VEL
LIN {X 0,Y 412.783,Z 453.815,A -85,B 0,C 180,E1 19384.436,E2 19384.436} C_VEL
LIN {X 0,Y 410.806,Z 472.967,A -85,B 0,C 180,E1 19383.456,E2 19383.456} C_VEL
LIN {X 0,Y 408.424,Z 492.567,A -85,B 0,C 180,E1 19382.173,E2 19382.173} C_VEL
LIN {X 0,Y 405.904,Z 511.244,A -85,B 0,C 180,E1 19380.658,E2 19380.658} C_VEL
LIN {X 0,Y 403.448,Z 528.391,A -85,B 0,C 180,E1 19378.975,E2 19378.975} C_VEL
LIN {X 0,Y 400.958,Z 545.305,A -85,B 0,C 180,E1 19376.992,E2 19376.992} C_VEL
LIN {X 0,Y 398.617,Z 561.219,A -85,B 0,C 180,E1 19374.765,E2 19374.765} C_VEL
LIN {X 0,Y 396.603,Z 575.565,A -85,B 0,C 180,E1 19372.377,E2 19372.377} C_VEL
LIN {X 0,Y 395.048,Z 587.741,A -85,B 0,C 180,E1 19369.98,E2 19369.98} C_VEL
LIN {X 0,Y 393.759,Z 599.216,A -85,B 0,C 180,E1 19367.284,E2 19367.284} C_VEL
LIN {X 0,Y 392.871,Z 609.092,A -85,B 0,C 180,E1 19364.443,E2 19364.443} C_VEL
LIN {X 0,Y 392.371,Z 616.941,A -85,B 0,C 180,E1 19361.615,E2 19361.615} C_VEL
LIN {X 0,Y 392.149,Z 622.974,A -85,B 0,C 180,E1 19358.801,E2 19358.801} C_VEL
LIN {X 0,Y 392.096,Z 627.483,A -85,B 0,C 180,E1 19355.855,E2 19355.855} C_VEL
LIN {X 0,Y 392.117,Z 630.105,A -85,B 0,C 180,E1 19353.07,E2 19353.07} C_VEL
LIN {X 0,Y 392.137,Z 631.041,A -85,B 0,C 180,E1 19350.439,E2 19350.439} C_VEL
LIN {X 0,Y 392.123,Z 630.478,A -85,B 0,C 180,E1 19347.663,E2 19347.663} C_VEL
LIN {X 0,Y 392.096,Z 628.348,A -85,B 0,C 180,E1 19344.88,E2 19344.88} C_VEL
LIN {X 0,Y 392.121,Z 624.564,A -85,B 0,C 180,E1 19342.087,E2 19342.087} C_VEL
LIN {X 0,Y 392.278,Z 619.037,A -85,B 0,C 180,E1 19339.278,E2 19339.278} C_VEL
LIN {X 0,Y 392.67,Z 611.739,A -85,B 0,C 180,E1 19336.453,E2 19336.453} C_VEL
LIN {X 0,Y 393.433,Z 602.512,A -85,B 0,C 180,E1 19333.616,E2 19333.616} C_VEL
LIN {X 0,Y 394.562,Z 591.783,A -85,B 0,C 180,E1 19330.92,E2 19330.92} C_VEL
LIN {X 0,Y 396.072,Z 579.623,A -85,B 0,C 180,E1 19328.374,E2 19328.374} C_VEL
LIN {X 0,Y 397.942,Z 566.019,A -85,B 0,C 180,E1 19325.982,E2 19325.982} C_VEL
LIN {X 0,Y 400.198,Z 550.403,A -85,B 0,C 180,E1 19323.676,E2 19323.676} C_VEL
LIN {X 0,Y 402.582,Z 534.322,A -85,B 0,C 180,E1 19321.683,E2 19321.683} C_VEL
LIN {X 0,Y 405.065,Z 516.994,A -85,B 0,C 180,E1 19319.878,E2 19319.878} C_VEL
LIN {X 0,Y 407.661,Z 498.163,A -85,B 0,C 180,E1 19318.259,E2 19318.259} C_VEL
LIN {X 0,Y 410.101,Z 478.664,A -85,B 0,C 180,E1 19316.899,E2 19316.899} C_VEL
LIN {X 0,Y 412.326,Z 458.301,A -85,B 0,C 180,E1 19315.781,E2 19315.781} C_VEL
LIN {X 0,Y 414.155,Z 437.912,A -85,B 0,C 180,E1 19314.936,E2 19314.936} C_VEL
LIN {X 0,Y 415.55,Z 417.114,A -85,B 0,C 180,E1 19314.332,E2 19314.332} C_VEL
LIN {X 0,Y 422.018,Z 213.372,A -85,B 0,C 180,E1 19310.428,E2 19310.428} C_VEL
LIN {X 0,Y 422.426,Z 194.517,A -85,B 0,C 180,E1 19310.055,E2 19310.055} C_VEL
LIN {X 0,Y 420.333,Z 178.648,A -85,B 0,C 180,E1 19309.49,E2 19309.49} C_VEL
LIN {X 0,Y 412.762,Z 164.898,A -85,B 0,C 180,E1 19308.356,E2 19308.356} C_VEL
LIN {X 0,Y 405.586,Z 147.073,A -85,B 0,C 180,E1 19305.565,E2 19305.565} C_VEL
LIN {X 0,Y 398.757,Z 132.071,A -85,B 0,C 180,E1 19302.933,E2 19302.933} C_VEL
LIN {X 0,Y 395.256,Z 124.531,A -85,B 0,C 180,E1 19301.511,E2 19301.511} C_VEL
LIN {X 0,Y 393.764,Z 121.675,A -85,B 0,C 180,E1 19300.929,E2 19300.929} C_VEL
LIN {X 0,Y 393.521,Z 120.433,A -85,B 0,C 180,E1 19300.695,E2 19300.695} C_VEL
LIN {X 0,Y 393.512,Z 120.421,A -85,B 0,C 180,E1 19296.837,E2 19296.837} C_VEL
LIN {X 0,Y 393.514,Z 120.448,A -85,B 0,C 180,E1 19292.938,E2 19292.938} C_VEL
LIN {X 0,Y 393.511,Z 120.449,A -85,B 0,C 180,E1 19289.032,E2 19289.032} C_VEL
LIN {X 0,Y 393.509,Z 120.457,A -85,B 0,C 180,E1 19285.108,E2 19285.108} C_VEL
LIN {X 0,Y 393.509,Z 120.467,A -85,B 0,C 180,E1 19281.149,E2 19281.149} C_VEL
LIN {X 0,Y 393.508,Z 120.462,A -85,B 0,C 180,E1 19277.142,E2 19277.142} C_VEL
LIN {X 0,Y 393.502,Z 120.44,A -85,B 0,C 180,E1 19273.219,E2 19273.219} C_VEL
LIN {X 0,Y 393.506,Z 120.465,A -85,B 0,C 180,E1 19269.211,E2 19269.211} C_VEL
LIN {X 0,Y 393.503,Z 120.462,A -85,B 0,C 180,E1 19265.248,E2 19265.248} C_VEL
LIN {X 0,Y 393.499,Z 120.441,A -85,B 0,C 180,E1 19261.31,E2 19261.31} C_VEL
LIN {X 0,Y 393.502,Z 120.467,A -85,B 0,C 180,E1 19257.378,E2 19257.378} C_VEL
LIN {X 0,Y 393.496,Z 120.451,A -85,B 0,C 180,E1 19253.434,E2 19253.434} C_VEL
LIN {X 0,Y 393.497,Z 120.451,A -85,B 0,C 180,E1 19249.458,E2 19249.458} C_VEL
LIN {X 0,Y 393.497,Z 120.468,A -85,B 0,C 180,E1 19245.43,E2 19245.43} C_VEL
LIN {X 0,Y 393.498,Z 120.45,A -85,B 0,C 180,E1 19241.397,E2 19241.397} C_VEL
LIN {X 0,Y 393.495,Z 120.448,A -85,B 0,C 180,E1 19237.437,E2 19237.437} C_VEL
LIN {X 0,Y 393.499,Z 120.466,A -85,B 0,C 180,E1 19233.43,E2 19233.43} C_VEL
LIN {X 0,Y 393.494,Z 120.467,A -85,B 0,C 180,E1 19229.471,E2 19229.471} C_VEL
LIN {X 0,Y 393.496,Z 120.464,A -85,B 0,C 180,E1 19225.484,E2 19225.484} C_VEL
LIN {X 0,Y 393.493,Z 120.464,A -85,B 0,C 180,E1 19221.498,E2 19221.498} C_VEL
LIN {X 0,Y 393.491,Z 120.468,A -85,B 0,C 180,E1 19217.672,E2 19217.672} C_VEL
LIN {X 0,Y 393.536,Z 120.589,A -85,B 0,C 180,E1 19215.029,E2 19215.029} C_VEL
LIN {X 0,Y 395.067,Z 124.312,A -85,B 0,C 180,E1 19214.255,E2 19214.255} C_VEL
LIN {X 0,Y 401.524,Z 139.414,A -85,B 0,C 180,E1 19211.233,E2 19211.233} C_VEL
LIN {X 0,Y 407.805,Z 155.623,A -85,B 0,C 180,E1 19208.318,E2 19208.318} C_VEL
LIN {X 0,Y 413.66,Z 172.773,A -85,B 0,C 180,E1 19205.545,E2 19205.545} C_VEL
LIN {X 0,Y 414.678,Z 175.629,A -85,B 0,C 180,E1 19205.361,E2 19205.361} C_VEL
LIN {X 0,Y 420.318,Z 209.823,A -85,B 0,C 180,E1 19204.074,E2 19204.074} C_VEL
LIN {X 0,Y 416.274,Z 392.597,A -85,B 0,C 180,E1 19200.977,E2 19200.977} C_VEL
LIN {X 0,Y 415.229,Z 411.804,A -85,B 0,C 180,E1 19200.402,E2 19200.402} C_VEL
LIN {X 0,Y 413.781,Z 429.854,A -85,B 0,C 180,E1 19199.613,E2 19199.613} C_VEL
LIN {X 0,Y 411.859,Z 447.675,A -85,B 0,C 180,E1 19198.57,E2 19198.57} C_VEL
LIN {X 0,Y 409.527,Z 465.278,A -85,B 0,C 180,E1 19197.243,E2 19197.243} C_VEL
LIN {X 0,Y 407.008,Z 481.654,A -85,B 0,C 180,E1 19195.694,E2 19195.694} C_VEL
LIN {X 0,Y 404.5,Z 496.334,A -85,B 0,C 180,E1 19193.991,E2 19193.991} C_VEL
LIN {X 0,Y 402.036,Z 509.819,A -85,B 0,C 180,E1 19192.092,E2 19192.092} C_VEL
LIN {X 0,Y 400.131,Z 515.067,A -85,B 0,C 180,E1 19191.315,E2 19191.315} C_VEL
LIN {X 0,Y 392.105,Z 527.682,A -85,B 0,C 180,E1 19189.361,E2 19189.361} C_VEL
LIN {X 0,Y 390.304,Z 532.061,A -85,B 0,C 180,E1 19188.469,E2 19188.469} C_VEL
LIN {X 0,Y 388.366,Z 541.938,A -85,B 0,C 180,E1 19185.989,E2 19185.989} C_VEL
LIN {X 0,Y 386.789,Z 550.499,A -85,B 0,C 180,E1 19183.3,E2 19183.3} C_VEL
LIN {X 0,Y 385.693,Z 557.165,A -85,B 0,C 180,E1 19180.605,E2 19180.605} C_VEL
LIN {X 0,Y 384.968,Z 562.384,A -85,B 0,C 180,E1 19177.761,E2 19177.761} C_VEL
LIN {X 0,Y 384.568,Z 565.891,A -85,B 0,C 180,E1 19174.921,E2 19174.921} C_VEL
LIN {X 0,Y 384.397,Z 567.803,A -85,B 0,C 180,E1 19172.086,E2 19172.086} C_VEL
LIN {X 0,Y 384.365,Z 568.167,A -85,B 0,C 180,E1 19169.105,E2 19169.105} C_VEL
LIN {X 0,Y 384.476,Z 566.85,A -85,B 0,C 180,E1 19166.122,E2 19166.122} C_VEL
LIN {X 0,Y 384.778,Z 563.99,A -85,B 0,C 180,E1 19163.284,E2 19163.284} C_VEL
LIN {X 0,Y 385.379,Z 559.338,A -85,B 0,C 180,E1 19160.37,E2 19160.37} C_VEL
LIN {X 0,Y 386.339,Z 553.156,A -85,B 0,C 180,E1 19157.595,E2 19157.595} C_VEL
LIN {X 0,Y 387.738,Z 545.325,A -85,B 0,C 180,E1 19154.902,E2 19154.902} C_VEL
LIN {X 0,Y 389.525,Z 536.031,A -85,B 0,C 180,E1 19152.368,E2 19152.368} C_VEL
LIN {X 0,Y 391.756,Z 524.936,A -85,B 0,C 180,E1 19149.923,E2 19149.923} C_VEL
LIN {X 0,Y 394.131,Z 513.118,A -85,B 0,C 180,E1 19147.79,E2 19147.79} C_VEL
LIN {X 0,Y 396.797,Z 499.394,A -85,B 0,C 180,E1 19145.748,E2 19145.748} C_VEL
LIN {X 0,Y 399.449,Z 484.885,A -85,B 0,C 180,E1 19143.977,E2 19143.977} C_VEL
LIN {X 0,Y 402.1,Z 468.76,A -85,B 0,C 180,E1 19142.37,E2 19142.37} C_VEL
LIN {X 0,Y 404.512,Z 451.904,A -85,B 0,C 180,E1 19141.022,E2 19141.022} C_VEL
LIN {X 0,Y 406.644,Z 433.897,A -85,B 0,C 180,E1 19139.893,E2 19139.893} C_VEL
LIN {X 0,Y 408.312,Z 415.375,A -85,B 0,C 180,E1 19139.022,E2 19139.022} C_VEL
LIN {X 0,Y 409.48,Z 396.354,A -85,B 0,C 180,E1 19138.399,E2 19138.399} C_VEL
LIN {X 0,Y 410.238,Z 370.43,A -85,B 0,C 180,E1 19137.894,E2 19137.894} C_VEL
LIN {X 0,Y 413.862,Z 209.782,A -85,B 0,C 180,E1 19135.144,E2 19135.144} C_VEL
LIN {X 0,Y 408.446,Z 177.764,A -85,B 0,C 180,E1 19133.885,E2 19133.885} C_VEL
LIN {X 0,Y 405.708,Z 172.726,A -85,B 0,C 180,E1 19133.459,E2 19133.459} C_VEL
LIN {X 0,Y 399.808,Z 155.789,A -85,B 0,C 180,E1 19130.603,E2 19130.603} C_VEL
LIN {X 0,Y 393.659,Z 140.145,A -85,B 0,C 180,E1 19127.656,E2 19127.656} C_VEL
LIN {X 0,Y 388.3,Z 128.07,A -85,B 0,C 180,E1 19125.126,E2 19125.126} C_VEL
LIN {X 0,Y 386.941,Z 124.97,A -85,B 0,C 180,E1 19124.449,E2 19124.449} C_VEL
LIN {X 0,Y 385.624,Z 121.436,A -85,B 0,C 180,E1 19123.663,E2 19123.663} C_VEL
LIN {X 0,Y 385.634,Z 121.497,A -85,B 0,C 180,E1 19121.529,E2 19121.529} C_VEL
LIN {X 0,Y 395.648,Z 147.706,A -85,B 0,C 180,E1 19117.956,E2 19117.956} C_VEL
LIN {X 0,Y 403.088,Z 169.463,A -85,B 0,C 180,E1 19115.181,E2 19115.181} C_VEL
LIN {X 0,Y 402.308,Z 186.461,A -85,B 0,C 180,E1 19113.663,E2 19113.663} C_VEL
LIN {X 0,Y 404.993,Z 208.177,A -85,B 0,C 180,E1 19112.898,E2 19112.898} C_VEL
LIN {X 0,Y 398.261,Z 398.142,A -85,B 0,C 180,E1 19108.669,E2 19108.669} C_VEL
LIN {X 0,Y 397.358,Z 417.483,A -85,B 0,C 180,E1 19107.967,E2 19107.967} C_VEL
LIN {X 0,Y 396.165,Z 436.388,A -85,B 0,C 180,E1 19107.01,E2 19107.01} C_VEL
LIN {X 0,Y 394.767,Z 454.377,A -85,B 0,C 180,E1 19105.826,E2 19105.826} C_VEL
LIN {X 0,Y 393.155,Z 472.422,A -85,B 0,C 180,E1 19104.33,E2 19104.33} C_VEL
LIN {X 0,Y 391.566,Z 488.569,A -85,B 0,C 180,E1 19102.68,E2 19102.68} C_VEL
LIN {X 0,Y 389.985,Z 503.721,A -85,B 0,C 180,E1 19100.799,E2 19100.799} C_VEL
LIN {X 0,Y 388.512,Z 517.48,A -85,B 0,C 180,E1 19098.723,E2 19098.723} C_VEL
LIN {X 0,Y 387.234,Z 529.63,A -85,B 0,C 180,E1 19096.501,E2 19096.501} C_VEL
LIN {X 0,Y 386.231,Z 539.844,A -85,B 0,C 180,E1 19094.237,E2 19094.237} C_VEL
LIN {X 0,Y 385.453,Z 548.696,A -85,B 0,C 180,E1 19091.825,E2 19091.825} C_VEL
LIN {X 0,Y 384.905,Z 556.109,A -85,B 0,C 180,E1 19089.269,E2 19089.269} C_VEL
LIN {X 0,Y 384.572,Z 561.989,A -85,B 0,C 180,E1 19086.569,E2 19086.569} C_VEL
LIN {X 0,Y 384.424,Z 565.823,A -85,B 0,C 180,E1 19084.027,E2 19084.027} C_VEL
LIN {X 0,Y 384.382,Z 568.172,A -85,B 0,C 180,E1 19081.342,E2 19081.342} C_VEL
LIN {X 0,Y 384.433,Z 568.805,A -85,B 0,C 180,E1 19078.659,E2 19078.659} C_VEL
LIN {X 0,Y 384.585,Z 567.726,A -85,B 0,C 180,E1 19075.975,E2 19075.975} C_VEL
LIN {X 0,Y 384.877,Z 564.918,A -85,B 0,C 180,E1 19073.287,E2 19073.287} C_VEL
LIN {X 0,Y 385.347,Z 560.58,A -85,B 0,C 180,E1 19070.743,E2 19070.743} C_VEL
LIN {X 0,Y 386.088,Z 554.528,A -85,B 0,C 180,E1 19068.195,E2 19068.195} C_VEL
LIN {X 0,Y 387.145,Z 546.548,A -85,B 0,C 180,E1 19065.645,E2 19065.645} C_VEL
LIN {X 0,Y 388.476,Z 536.903,A -85,B 0,C 180,E1 19063.229,E2 19063.229} C_VEL
LIN {X 0,Y 390.026,Z 525.908,A -85,B 0,C 180,E1 19061,E2 19061} C_VEL
LIN {X 0,Y 391.916,Z 512.312,A -85,B 0,C 180,E1 19058.761,E2 19058.761} C_VEL
LIN {X 0,Y 393.748,Z 498.518,A -85,B 0,C 180,E1 19056.901,E2 19056.901} C_VEL
LIN {X 0,Y 395.65,Z 483.235,A -85,B 0,C 180,E1 19055.197,E2 19055.197} C_VEL
LIN {X 0,Y 397.452,Z 466.993,A -85,B 0,C 180,E1 19053.72,E2 19053.72} C_VEL
LIN {X 0,Y 399.215,Z 448.906,A -85,B 0,C 180,E1 19052.397,E2 19052.397} C_VEL
LIN {X 0,Y 400.76,Z 429.57,A -85,B 0,C 180,E1 19051.297,E2 19051.297} C_VEL
LIN {X 0,Y 402.041,Z 409.753,A -85,B 0,C 180,E1 19050.45,E2 19050.45} C_VEL
LIN {X 0,Y 404.233,Z 370.405,A -85,B 0,C 180,E1 19049.326,E2 19049.326} C_VEL
LIN {X 0,Y 409.897,Z 296.982,A -85,B 0,C 180,E1 19047.223,E2 19047.223} C_VEL
LIN {X 0,Y 418.66,Z 212.239,A -85,B 0,C 180,E1 19044.667,E2 19044.667} C_VEL
LIN {X 0,Y 418.272,Z 202.637,A -85,B 0,C 180,E1 19043.981,E2 19043.981} C_VEL
LIN {X 0,Y 420.951,Z 181.813,A -85,B 0,C 180,E1 19041.992,E2 19041.992} C_VEL
LIN {X 0,Y 419.676,Z 174.638,A -85,B 0,C 180,E1 19040.498,E2 19040.498} C_VEL
LIN {X 0,Y 418.335,Z 168.853,A -85,B 0,C 180,E1 19038.841,E2 19038.841} C_VEL
LIN {X 0,Y 417.457,Z 164.672,A -85,B 0,C 180,E1 19037.132,E2 19037.132} C_VEL
LIN {X 0,Y 417.005,Z 163.178,A -85,B 0,C 180,E1 19035.462,E2 19035.462} C_VEL
LIN {X 0,Y 415.771,Z 166.878,A -85,B 0,C 180,E1 19034.42,E2 19034.42} C_VEL
LIN {X 0,Y 414.964,Z 172.11,A -85,B 0,C 180,E1 19033.107,E2 19033.107} C_VEL
LIN {X 0,Y 414.839,Z 178.312,A -85,B 0,C 180,E1 19031.802,E2 19031.802} C_VEL
LIN {X 0,Y 414.749,Z 183.535,A -85,B 0,C 180,E1 19031.04,E2 19031.04} C_VEL
LIN {X 0,Y 416.159,Z 198.53,A -85,B 0,C 180,E1 19030.518,E2 19030.518} C_VEL
LIN {X 0,Y 409.042,Z 412.967,A -85,B 0,C 180,E1 19026.373,E2 19026.373} C_VEL
LIN {X 0,Y 407.659,Z 434.854,A -85,B 0,C 180,E1 19025.769,E2 19025.769} C_VEL
LIN {X 0,Y 405.779,Z 455.259,A -85,B 0,C 180,E1 19024.953,E2 19024.953} C_VEL
LIN {X 0,Y 403.638,Z 474.662,A -85,B 0,C 180,E1 19023.919,E2 19023.919} C_VEL
LIN {X 0,Y 401.218,Z 493.581,A -85,B 0,C 180,E1 19022.644,E2 19022.644} C_VEL
LIN {X 0,Y 398.5,Z 512.647,A -85,B 0,C 180,E1 19021.05,E2 19021.05} C_VEL
LIN {X 0,Y 395.727,Z 530.887,A -85,B 0,C 180,E1 19019.186,E2 19019.186} C_VEL
LIN {X 0,Y 393.06,Z 547.924,A -85,B 0,C 180,E1 19017.087,E2 19017.087} C_VEL
LIN {X 0,Y 390.668,Z 563.316,A -85,B 0,C 180,E1 19014.819,E2 19014.819} C_VEL
LIN {X 0,Y 388.603,Z 577.221,A -85,B 0,C 180,E1 19012.384,E2 19012.384} C_VEL
LIN {X 0,Y 386.931,Z 589.685,A -85,B 0,C 180,E1 19009.787,E2 19009.787} C_VEL
LIN {X 0,Y 385.659,Z 600.686,A -85,B 0,C 180,E1 19007.036,E2 19007.036} C_VEL
LIN {X 0,Y 384.828,Z 609.771,A -85,B 0,C 180,E1 19004.275,E2 19004.275} C_VEL
LIN {X 0,Y 384.345,Z 617.363,A -85,B 0,C 180,E1 19001.404,E2 19001.404} C_VEL
LIN {X 0,Y 384.14,Z 623.228,A -85,B 0,C 180,E1 18998.476,E2 18998.476} C_VEL
LIN {X 0,Y 384.114,Z 627.173,A -85,B 0,C 180,E1 18995.678,E2 18995.678} C_VEL
LIN {X 0,Y 384.146,Z 629.607,A -85,B 0,C 180,E1 18992.836,E2 18992.836} C_VEL
LIN {X 0,Y 384.176,Z 630.461,A -85,B 0,C 180,E1 18990.001,E2 18990.001} C_VEL
LIN {X 0,Y 384.146,Z 629.607,A -85,B 0,C 180,E1 18987.166,E2 18987.166} C_VEL
LIN {X 0,Y 384.114,Z 627.171,A -85,B 0,C 180,E1 18984.324,E2 18984.324} C_VEL
LIN {X 0,Y 384.142,Z 623.126,A -85,B 0,C 180,E1 18981.469,E2 18981.469} C_VEL
LIN {X 0,Y 384.347,Z 617.368,A -85,B 0,C 180,E1 18978.598,E2 18978.598} C_VEL
LIN {X 0,Y 384.831,Z 609.728,A -85,B 0,C 180,E1 18975.711,E2 18975.711} C_VEL
LIN {X 0,Y 385.658,Z 600.683,A -85,B 0,C 180,E1 18972.966,E2 18972.966} C_VEL
LIN {X 0,Y 386.974,Z 589.327,A -85,B 0,C 180,E1 18970.135,E2 18970.135} C_VEL
LIN {X 0,Y 388.75,Z 576.154,A -85,B 0,C 180,E1 18967.419,E2 18967.419} C_VEL
LIN {X 0,Y 390.95,Z 561.359,A -85,B 0,C 180,E1 18964.879,E2 18964.879} C_VEL
LIN {X 0,Y 393.408,Z 545.58,A -85,B 0,C 180,E1 18962.613,E2 18962.613} C_VEL
LIN {X 0,Y 395.922,Z 529.473,A -85,B 0,C 180,E1 18960.666,E2 18960.666} C_VEL
LIN {X 0,Y 398.59,Z 511.881,A -85,B 0,C 180,E1 18958.887,E2 18958.887} C_VEL
LIN {X 0,Y 401.221,Z 493.427,A -85,B 0,C 180,E1 18957.35,E2 18957.35} C_VEL
LIN {X 0,Y 403.695,Z 474.044,A -85,B 0,C 180,E1 18956.049,E2 18956.049} C_VEL
LIN {X 0,Y 405.846,Z 454.423,A -85,B 0,C 180,E1 18955.013,E2 18955.013} C_VEL
LIN {X 0,Y 407.69,Z 434.207,A -85,B 0,C 180,E1 18954.215,E2 18954.215} C_VEL
LIN {X 0,Y 409.028,Z 412.737,A -85,B 0,C 180,E1 18953.627,E2 18953.627} C_VEL
LIN {X 0,Y 416.177,Z 197.11,A -85,B 0,C 180,E1 18949.461,E2 18949.461} C_VEL
LIN {X 0,Y 414.297,Z 182.331,A -85,B 0,C 180,E1 18948.927,E2 18948.927} C_VEL
LIN {X 0,Y 404.616,Z 164.629,A -85,B 0,C 180,E1 18947.385,E2 18947.385} C_VEL
LIN {X 0,Y 397.55,Z 147.504,A -85,B 0,C 180,E1 18944.563,E2 18944.563} C_VEL
LIN {X 0,Y 391.261,Z 133.688,A -85,B 0,C 180,E1 18942.031,E2 18942.031} C_VEL
LIN {X 0,Y 386.907,Z 124.873,A -85,B 0,C 180,E1 18940.245,E2 18940.245} C_VEL
LIN {X 0,Y 385.574,Z 121.393,A -85,B 0,C 180,E1 18939.539,E2 18939.539} C_VEL
LIN {X 0,Y 385.585,Z 121.443,A -85,B 0,C 180,E1 18935.693,E2 18935.693} C_VEL
LIN {X 0,Y 385.587,Z 121.445,A -85,B 0,C 180,E1 18931.733,E2 18931.733} C_VEL
LIN {X 0,Y 385.593,Z 121.438,A -85,B 0,C 180,E1 18927.846,E2 18927.846} C_VEL
LIN {X 0,Y 385.587,Z 121.432,A -85,B 0,C 180,E1 18923.861,E2 18923.861} C_VEL
LIN {X 0,Y 385.597,Z 121.439,A -85,B 0,C 180,E1 18920.015,E2 18920.015} C_VEL
LIN {X 0,Y 385.59,Z 121.455,A -85,B 0,C 180,E1 18915.954,E2 18915.954} C_VEL
LIN {X 0,Y 385.595,Z 121.431,A -85,B 0,C 180,E1 18912.124,E2 18912.124} C_VEL
LIN {X 0,Y 385.599,Z 121.43,A -85,B 0,C 180,E1 18908.199,E2 18908.199} C_VEL
LIN {X 0,Y 385.594,Z 121.457,A -85,B 0,C 180,E1 18904.163,E2 18904.163} C_VEL
LIN {X 0,Y 385.589,Z 121.428,A -85,B 0,C 180,E1 18900.148,E2 18900.148} C_VEL
LIN {X 0,Y 385.592,Z 121.441,A -85,B 0,C 180,E1 18896.283,E2 18896.283} C_VEL
LIN {X 0,Y 385.594,Z 121.45,A -85,B 0,C 180,E1 18892.25,E2 18892.25} C_VEL
LIN {X 0,Y 385.59,Z 121.426,A -85,B 0,C 180,E1 18888.331,E2 18888.331} C_VEL
LIN {X 0,Y 385.595,Z 121.447,A -85,B 0,C 180,E1 18884.355,E2 18884.355} C_VEL
LIN {X 0,Y 385.586,Z 121.45,A -85,B 0,C 180,E1 18880.299,E2 18880.299} C_VEL
LIN {X 0,Y 385.594,Z 121.428,A -85,B 0,C 180,E1 18876.463,E2 18876.463} C_VEL
LIN {X 0,Y 385.596,Z 121.432,A -85,B 0,C 180,E1 18872.473,E2 18872.473} C_VEL
LIN {X 0,Y 385.598,Z 121.448,A -85,B 0,C 180,E1 18868.548,E2 18868.548} C_VEL
LIN {X 0,Y 385.586,Z 121.455,A -85,B 0,C 180,E1 18864.489,E2 18864.489} C_VEL
LIN {X 0,Y 385.594,Z 121.455,A -85,B 0,C 180,E1 18860.558,E2 18860.558} C_VEL
LIN {X 0,Y 385.585,Z 121.447,A -85,B 0,C 180,E1 18856.556,E2 18856.556} C_VEL
LIN {X 0,Y 385.57,Z 121.512,A -85,B 0,C 180,E1 18856.18,E2 18856.18} C_VEL
LIN {X 0,Y 386.701,Z 124.684,A -85,B 0,C 180,E1 18855.516,E2 18855.516} C_VEL
LIN {X 0,Y 387.727,Z 126.764,A -85,B 0,C 180,E1 18855.042,E2 18855.042} C_VEL
LIN {X 0,Y 392.738,Z 138.261,A -85,B 0,C 180,E1 18852.624,E2 18852.624} C_VEL
LIN {X 0,Y 398.582,Z 152.636,A -85,B 0,C 180,E1 18849.86,E2 18849.86} C_VEL
LIN {X 0,Y 404.503,Z 169.126,A -85,B 0,C 180,E1 18847.022,E2 18847.022} C_VEL
LIN {X 0,Y 405.967,Z 173.304,A -85,B 0,C 180,E1 18846.387,E2 18846.387} C_VEL
LIN {X 0,Y 408.64,Z 178.656,A -85,B 0,C 180,E1 18845.968,E2 18845.968} C_VEL
LIN {X 0,Y 413.91,Z 211.25,A -85,B 0,C 180,E1 18844.716,E2 18844.716} C_VEL
LIN {X 0,Y 409.618,Z 392.99,A -85,B 0,C 180,E1 18841.59,E2 18841.59} C_VEL
LIN {X 0,Y 408.516,Z 412.26,A -85,B 0,C 180,E1 18841.005,E2 18841.005} C_VEL
LIN {X 0,Y 407.054,Z 429.742,A -85,B 0,C 180,E1 18840.234,E2 18840.234} C_VEL
LIN {X 0,Y 405.044,Z 447.684,A -85,B 0,C 180,E1 18839.177,E2 18839.177} C_VEL
LIN {X 0,Y 402.68,Z 464.879,A -85,B 0,C 180,E1 18837.877,E2 18837.877} C_VEL
LIN {X 0,Y 400.076,Z 481.183,A -85,B 0,C 180,E1 18836.333,E2 18836.333} C_VEL
LIN {X 0,Y 397.327,Z 496.579,A -85,B 0,C 180,E1 18834.532,E2 18834.532} C_VEL
LIN {X 0,Y 394.591,Z 510.78,A -85,B 0,C 180,E1 18832.495,E2 18832.495} C_VEL
LIN {X 0,Y 392.071,Z 523.367,A -85,B 0,C 180,E1 18830.292,E2 18830.292} C_VEL
LIN {X 0,Y 390.304,Z 532.061,A -85,B 0,C 180,E1 18828.469,E2 18828.469} C_VEL
LIN {X 0,Y 388.55,Z 536.3,A -85,B 0,C 180,E1 18827.547,E2 18827.547} C_VEL
LIN {X 0,Y 381.266,Z 545.723,A -85,B 0,C 180,E1 18825.337,E2 18825.337} C_VEL
LIN {X 0,Y 379.409,Z 549.084,A -85,B 0,C 180,E1 18824.318,E2 18824.318} C_VEL
LIN {X 0,Y 379.297,Z 549.518,A -85,B 0,C 180,E1 18824.165,E2 18824.165} C_VEL
LIN {X 0,Y 378.035,Z 556.509,A -85,B 0,C 180,E1 18821.44,E2 18821.44} C_VEL
LIN {X 0,Y 377.173,Z 562.097,A -85,B 0,C 180,E1 18818.536,E2 18818.536} C_VEL
LIN {X 0,Y 376.677,Z 565.953,A -85,B 0,C 180,E1 18815.635,E2 18815.635} C_VEL
LIN {X 0,Y 376.447,Z 568.201,A -85,B 0,C 180,E1 18812.739,E2 18812.739} C_VEL
LIN {X 0,Y 376.393,Z 568.917,A -85,B 0,C 180,E1 18809.847,E2 18809.847} C_VEL
LIN {X 0,Y 376.466,Z 568.019,A -85,B 0,C 180,E1 18806.802,E2 18806.802} C_VEL
LIN {X 0,Y 376.728,Z 565.595,A -85,B 0,C 180,E1 18803.905,E2 18803.905} C_VEL
LIN {X 0,Y 377.304,Z 561.257,A -85,B 0,C 180,E1 18800.85,E2 18800.85} C_VEL
LIN {X 0,Y 378.249,Z 555.338,A -85,B 0,C 180,E1 18797.945,E2 18797.945} C_VEL
LIN {X 0,Y 379.659,Z 547.741,A -85,B 0,C 180,E1 18795.134,E2 18795.134} C_VEL
LIN {X 0,Y 381.515,Z 538.531,A -85,B 0,C 180,E1 18792.458,E2 18792.458} C_VEL
LIN {X 0,Y 383.696,Z 528.217,A -85,B 0,C 180,E1 18790.039,E2 18790.039} C_VEL
LIN {X 0,Y 386.19,Z 516.522,A -85,B 0,C 180,E1 18787.789,E2 18787.789} C_VEL
LIN {X 0,Y 389.009,Z 502.847,A -85,B 0,C 180,E1 18785.635,E2 18785.635} C_VEL
LIN {X 0,Y 391.888,Z 488.008,A -85,B 0,C 180,E1 18783.725,E2 18783.725} C_VEL
LIN {X 0,Y 394.568,Z 472.83,A -85,B 0,C 180,E1 18782.125,E2 18782.125} C_VEL
LIN {X 0,Y 397.191,Z 455.874,A -85,B 0,C 180,E1 18780.684,E2 18780.684} C_VEL
LIN {X 0,Y 399.4,Z 438.9,A -85,B 0,C 180,E1 18779.539,E2 18779.539} C_VEL
LIN {X 0,Y 401.293,Z 420.225,A -85,B 0,C 180,E1 18778.58,E2 18778.58} C_VEL
LIN {X 0,Y 402.646,Z 401.302,A -85,B 0,C 180,E1 18777.889,E2 18777.889} C_VEL
LIN {X 0,Y 403.435,Z 381.304,A -85,B 0,C 180,E1 18777.433,E2 18777.433} C_VEL
LIN {X 0,Y 407.516,Z 211.161,A -85,B 0,C 180,E1 18774.48,E2 18774.48} C_VEL
LIN {X 0,Y 402.568,Z 181.535,A -85,B 0,C 180,E1 18773.285,E2 18773.285} C_VEL
LIN {X 0,Y 397.704,Z 172.47,A -85,B 0,C 180,E1 18772.485,E2 18772.485} C_VEL
LIN {X 0,Y 391.545,Z 155.224,A -85,B 0,C 180,E1 18769.439,E2 18769.439} C_VEL
LIN {X 0,Y 385.635,Z 140.694,A -85,B 0,C 180,E1 18766.55,E2 18766.55} C_VEL
LIN {X 0,Y 380.926,Z 130.057,A -85,B 0,C 180,E1 18764.227,E2 18764.227} C_VEL
LIN {X 0,Y 379.024,Z 125.96,A -85,B 0,C 180,E1 18763.273,E2 18763.273} C_VEL
LIN {X 0,Y 377.674,Z 122.431,A -85,B 0,C 180,E1 18762.462,E2 18762.462} C_VEL
LIN {X 0,Y 377.683,Z 122.465,A -85,B 0,C 180,E1 18762.255,E2 18762.255} C_VEL
LIN {X 0,Y 387.531,Z 147.971,A -85,B 0,C 180,E1 18758.695,E2 18758.695} C_VEL
LIN {X 0,Y 394.987,Z 169.349,A -85,B 0,C 180,E1 18755.899,E2 18755.899} C_VEL
LIN {X 0,Y 395.89,Z 172.514,A -85,B 0,C 180,E1 18755.513,E2 18755.513} C_VEL
LIN {X 0,Y 395.224,Z 186.991,A -85,B 0,C 180,E1 18754.221,E2 18754.221} C_VEL
LIN {X 0,Y 397.908,Z 209.235,A -85,B 0,C 180,E1 18753.418,E2 18753.418} C_VEL
LIN {X 0,Y 390.834,Z 398.773,A -85,B 0,C 180,E1 18749.094,E2 18749.094} C_VEL
LIN {X 0,Y 389.887,Z 418.129,A -85,B 0,C 180,E1 18748.374,E2 18748.374} C_VEL
LIN {X 0,Y 388.671,Z 436.683,A -85,B 0,C 180,E1 18747.418,E2 18747.418} C_VEL
LIN {X 0,Y 387.206,Z 454.847,A -85,B 0,C 180,E1 18746.204,E2 18746.204} C_VEL
LIN {X 0,Y 385.531,Z 472.924,A -85,B 0,C 180,E1 18744.68,E2 18744.68} C_VEL
LIN {X 0,Y 383.876,Z 489.106,A -85,B 0,C 180,E1 18742.998,E2 18742.998} C_VEL
LIN {X 0,Y 382.231,Z 504.294,A -85,B 0,C 180,E1 18741.081,E2 18741.081} C_VEL
LIN {X 0,Y 380.725,Z 517.847,A -85,B 0,C 180,E1 18739.005,E2 18739.005} C_VEL
LIN {X 0,Y 379.364,Z 530.274,A -85,B 0,C 180,E1 18736.696,E2 18736.696} C_VEL
LIN {X 0,Y 378.32,Z 540.518,A -85,B 0,C 180,E1 18734.385,E2 18734.385} C_VEL
LIN {X 0,Y 377.51,Z 549.398,A -85,B 0,C 180,E1 18731.923,E2 18731.923} C_VEL
LIN {X 0,Y 376.941,Z 556.835,A -85,B 0,C 180,E1 18729.312,E2 18729.312} C_VEL
LIN {X 0,Y 376.596,Z 562.727,A -85,B 0,C 180,E1 18726.556,E2 18726.556} C_VEL
LIN {X 0,Y 376.443,Z 566.737,A -85,B 0,C 180,E1 18723.808,E2 18723.808} C_VEL
LIN {X 0,Y 376.41,Z 568.895,A -85,B 0,C 180,E1 18721.218,E2 18721.218} C_VEL
LIN {X 0,Y 376.467,Z 569.525,A -85,B 0,C 180,E1 18718.631,E2 18718.631} C_VEL
LIN {X 0,Y 376.634,Z 568.521,A -85,B 0,C 180,E1 18715.89,E2 18715.89} C_VEL
LIN {X 0,Y 376.959,Z 565.776,A -85,B 0,C 180,E1 18713.145,E2 18713.145} C_VEL
LIN {X 0,Y 377.478,Z 561.522,A -85,B 0,C 180,E1 18710.548,E2 18710.548} C_VEL
LIN {X 0,Y 378.283,Z 555.517,A -85,B 0,C 180,E1 18707.948,E2 18707.948} C_VEL
LIN {X 0,Y 379.434,Z 547.621,A -85,B 0,C 180,E1 18705.347,E2 18705.347} C_VEL
LIN {X 0,Y 380.865,Z 538.145,A -85,B 0,C 180,E1 18702.901,E2 18702.901} C_VEL
LIN {X 0,Y 382.545,Z 527.161,A -85,B 0,C 180,E1 18700.614,E2 18700.614} C_VEL
LIN {X 0,Y 384.423,Z 514.655,A -85,B 0,C 180,E1 18698.486,E2 18698.486} C_VEL
LIN {X 0,Y 386.539,Z 500.056,A -85,B 0,C 180,E1 18696.444,E2 18696.444} C_VEL
LIN {X 0,Y 388.659,Z 484.207,A -85,B 0,C 180,E1 18694.638,E2 18694.638} C_VEL
LIN {X 0,Y 390.608,Z 468.168,A -85,B 0,C 180,E1 18693.141,E2 18693.141} C_VEL
LIN {X 0,Y 392.602,Z 449.143,A -85,B 0,C 180,E1 18691.726,E2 18691.726} C_VEL
LIN {X 0,Y 394.287,Z 429.958,A -85,B 0,C 180,E1 18690.614,E2 18690.614} C_VEL
LIN {X 0,Y 395.701,Z 410.014,A -85,B 0,C 180,E1 18689.745,E2 18689.745} C_VEL
LIN {X 0,Y 398.951,Z 360.822,A -85,B 0,C 180,E1 18688.292,E2 18688.292} C_VEL
LIN {X 0,Y 405.543,Z 287.863,A -85,B 0,C 180,E1 18686.09,E2 18686.09} C_VEL
LIN {X 0,Y 414.121,Z 213.419,A -85,B 0,C 180,E1 18683.735,E2 18683.735} C_VEL
LIN {X 0,Y 413.989,Z 204.238,A -85,B 0,C 180,E1 18683.032,E2 18683.032} C_VEL
LIN {X 0,Y 416.632,Z 186.588,A -85,B 0,C 180,E1 18681.306,E2 18681.306} C_VEL
LIN {X 0,Y 415.639,Z 179.495,A -85,B 0,C 180,E1 18679.692,E2 18679.692} C_VEL
LIN {X 0,Y 414.765,Z 174.591,A -85,B 0,C 180,E1 18678.106,E2 18678.106} C_VEL
LIN {X 0,Y 414.447,Z 171.835,A -85,B 0,C 180,E1 18676.753,E2 18676.753} C_VEL
LIN {X 0,Y 414.264,Z 170.917,A -85,B 0,C 180,E1 18675.651,E2 18675.651} C_VEL
LIN {X 0,Y 412.468,Z 177.417,A -85,B 0,C 180,E1 18673.892,E2 18673.892} C_VEL
LIN {X 0,Y 411.81,Z 184.569,A -85,B 0,C 180,E1 18672.368,E2 18672.368} C_VEL
LIN {X 0,Y 411.584,Z 187.614,A -85,B 0,C 180,E1 18671.918,E2 18671.918} C_VEL
LIN {X 0,Y 409.854,Z 198.411,A -85,B 0,C 180,E1 18671.205,E2 18671.205} C_VEL
LIN {X 0,Y 402.398,Z 412.862,A -85,B 0,C 180,E1 18667.006,E2 18667.006} C_VEL
LIN {X 0,Y 400.949,Z 434.789,A -85,B 0,C 180,E1 18666.391,E2 18666.391} C_VEL
LIN {X 0,Y 398.957,Z 455.381,A -85,B 0,C 180,E1 18665.552,E2 18665.552} C_VEL
LIN {X 0,Y 396.64,Z 475.261,A -85,B 0,C 180,E1 18664.468,E2 18664.468} C_VEL
LIN {X 0,Y 394.041,Z 494.435,A -85,B 0,C 180,E1 18663.138,E2 18663.138} C_VEL
LIN {X 0,Y 391.321,Z 512.592,A -85,B 0,C 180,E1 18661.588,E2 18661.588} C_VEL
LIN {X 0,Y 388.438,Z 530.589,A -85,B 0,C 180,E1 18659.715,E2 18659.715} C_VEL
LIN {X 0,Y 385.706,Z 547.07,A -85,B 0,C 180,E1 18657.648,E2 18657.648} C_VEL
LIN {X 0,Y 383.153,Z 562.51,A -85,B 0,C 180,E1 18655.34,E2 18655.34} C_VEL
LIN {X 0,Y 380.952,Z 576.449,A -85,B 0,C 180,E1 18652.859,E2 18652.859} C_VEL
LIN {X 0,Y 379.161,Z 588.94,A -85,B 0,C 180,E1 18650.21,E2 18650.21} C_VEL
LIN {X 0,Y 377.79,Z 599.965,A -85,B 0,C 180,E1 18647.402,E2 18647.402} C_VEL
LIN {X 0,Y 376.898,Z 609.027,A -85,B 0,C 180,E1 18644.598,E2 18644.598} C_VEL
LIN {X 0,Y 376.374,Z 616.681,A -85,B 0,C 180,E1 18641.649,E2 18641.649} C_VEL
LIN {X 0,Y 376.158,Z 622.455,A -85,B 0,C 180,E1 18638.715,E2 18638.715} C_VEL
LIN {X 0,Y 376.128,Z 626.517,A -85,B 0,C 180,E1 18635.799,E2 18635.799} C_VEL
LIN {X 0,Y 376.168,Z 628.96,A -85,B 0,C 180,E1 18632.896,E2 18632.896} C_VEL
LIN {X 0,Y 376.202,Z 629.816,A -85,B 0,C 180,E1 18630.001,E2 18630.001} C_VEL
LIN {X 0,Y 376.171,Z 629.034,A -85,B 0,C 180,E1 18627.259,E2 18627.259} C_VEL
LIN {X 0,Y 376.131,Z 626.688,A -85,B 0,C 180,E1 18624.357,E2 18624.357} C_VEL
LIN {X 0,Y 376.151,Z 622.73,A -85,B 0,C 180,E1 18621.44,E2 18621.44} C_VEL
LIN {X 0,Y 376.357,Z 617.013,A -85,B 0,C 180,E1 18618.508,E2 18618.508} C_VEL
LIN {X 0,Y 376.863,Z 609.443,A -85,B 0,C 180,E1 18615.553,E2 18615.553} C_VEL
LIN {X 0,Y 377.73,Z 600.509,A -85,B 0,C 180,E1 18612.756,E2 18612.756} C_VEL
LIN {X 0,Y 379.117,Z 589.25,A -85,B 0,C 180,E1 18609.866,E2 18609.866} C_VEL
LIN {X 0,Y 380.832,Z 577.249,A -85,B 0,C 180,E1 18607.299,E2 18607.299} C_VEL
LIN {X 0,Y 383.003,Z 563.46,A -85,B 0,C 180,E1 18604.817,E2 18604.817} C_VEL
LIN {X 0,Y 385.533,Z 548.084,A -85,B 0,C 180,E1 18602.493,E2 18602.493} C_VEL
LIN {X 0,Y 388.305,Z 531.295,A -85,B 0,C 180,E1 18600.372,E2 18600.372} C_VEL
LIN {X 0,Y 391.186,Z 513.305,A -85,B 0,C 180,E1 18598.488,E2 18598.488} C_VEL
LIN {X 0,Y 394.025,Z 494.398,A -85,B 0,C 180,E1 18596.865,E2 18596.865} C_VEL
LIN {X 0,Y 396.575,Z 475.567,A -85,B 0,C 180,E1 18595.559,E2 18595.559} C_VEL
LIN {X 0,Y 398.863,Z 456.012,A -85,B 0,C 180,E1 18594.484,E2 18594.484} C_VEL
LIN {X 0,Y 400.902,Z 435.019,A -85,B 0,C 180,E1 18593.623,E2 18593.623} C_VEL
LIN {X 0,Y 402.349,Z 413.314,A -85,B 0,C 180,E1 18593.01,E2 18593.01} C_VEL
LIN {X 0,Y 409.796,Z 199.01,A -85,B 0,C 180,E1 18588.813,E2 18588.813} C_VEL
LIN {X 0,Y 408.221,Z 185.8,A -85,B 0,C 180,E1 18588.334,E2 18588.334} C_VEL
LIN {X 0,Y 396.717,Z 165.238,A -85,B 0,C 180,E1 18586.487,E2 18586.487} C_VEL
LIN {X 0,Y 389.94,Z 149.002,A -85,B 0,C 180,E1 18583.692,E2 18583.692} C_VEL
LIN {X 0,Y 383.67,Z 135.194,A -85,B 0,C 180,E1 18581.05,E2 18581.05} C_VEL
LIN {X 0,Y 379.454,Z 126.554,A -85,B 0,C 180,E1 18579.225,E2 18579.225} C_VEL
LIN {X 0,Y 377.853,Z 123.427,A -85,B 0,C 180,E1 18578.523,E2 18578.523} C_VEL
LIN {X 0,Y 377.666,Z 122.368,A -85,B 0,C 180,E1 18578.28,E2 18578.28} C_VEL
LIN {X 0,Y 377.671,Z 122.432,A -85,B 0,C 180,E1 18574.142,E2 18574.142} C_VEL
LIN {X 0,Y 377.667,Z 122.434,A -85,B 0,C 180,E1 18570.024,E2 18570.024} C_VEL
LIN {X 0,Y 377.665,Z 122.441,A -85,B 0,C 180,E1 18566.07,E2 18566.07} C_VEL
LIN {X 0,Y 377.667,Z 122.436,A -85,B 0,C 180,E1 18562.082,E2 18562.082} C_VEL
LIN {X 0,Y 377.656,Z 122.419,A -85,B 0,C 180,E1 18558.045,E2 18558.045} C_VEL
LIN {X 0,Y 377.658,Z 122.419,A -85,B 0,C 180,E1 18554.097,E2 18554.097} C_VEL
LIN {X 0,Y 377.653,Z 122.444,A -85,B 0,C 180,E1 18550.063,E2 18550.063} C_VEL
LIN {X 0,Y 377.649,Z 122.419,A -85,B 0,C 180,E1 18546.079,E2 18546.079} C_VEL
LIN {X 0,Y 377.649,Z 122.422,A -85,B 0,C 180,E1 18542.124,E2 18542.124} C_VEL
LIN {X 0,Y 377.652,Z 122.444,A -85,B 0,C 180,E1 18538.179,E2 18538.179} C_VEL
LIN {X 0,Y 377.639,Z 122.415,A -85,B 0,C 180,E1 18534.073,E2 18534.073} C_VEL
LIN {X 0,Y 377.649,Z 122.434,A -85,B 0,C 180,E1 18530.244,E2 18530.244} C_VEL
LIN {X 0,Y 377.645,Z 122.438,A -85,B 0,C 180,E1 18526.214,E2 18526.214} C_VEL
LIN {X 0,Y 377.645,Z 122.415,A -85,B 0,C 180,E1 18522.273,E2 18522.273} C_VEL
LIN {X 0,Y 377.641,Z 122.432,A -85,B 0,C 180,E1 18518.243,E2 18518.243} C_VEL
LIN {X 0,Y 377.637,Z 122.444,A -85,B 0,C 180,E1 18514.182,E2 18514.182} C_VEL
LIN {X 0,Y 377.636,Z 122.429,A -85,B 0,C 180,E1 18510.275,E2 18510.275} C_VEL
LIN {X 0,Y 377.643,Z 122.424,A -85,B 0,C 180,E1 18506.402,E2 18506.402} C_VEL
LIN {X 0,Y 377.636,Z 122.428,A -85,B 0,C 180,E1 18502.339,E2 18502.339} C_VEL
LIN {X 0,Y 377.649,Z 122.43,A -85,B 0,C 180,E1 18498.525,E2 18498.525} C_VEL
LIN {X 0,Y 377.625,Z 122.486,A -85,B 0,C 180,E1 18497.396,E2 18497.396} C_VEL
LIN {X 0,Y 378.844,Z 125.751,A -85,B 0,C 180,E1 18496.669,E2 18496.669} C_VEL
LIN {X 0,Y 383.119,Z 134.951,A -85,B 0,C 180,E1 18494.563,E2 18494.563} C_VEL
LIN {X 0,Y 389.115,Z 149.268,A -85,B 0,C 180,E1 18491.604,E2 18491.604} C_VEL
LIN {X 0,Y 395.083,Z 165.038,A -85,B 0,C 180,E1 18488.688,E2 18488.688} C_VEL
LIN {X 0,Y 397.918,Z 173.082,A -85,B 0,C 180,E1 18487.348,E2 18487.348} C_VEL
LIN {X 0,Y 402.813,Z 182.542,A -85,B 0,C 180,E1 18486.556,E2 18486.556} C_VEL
LIN {X 0,Y 407.551,Z 212.713,A -85,B 0,C 180,E1 18485.378,E2 18485.378} C_VEL
LIN {X 0,Y 403.02,Z 393.186,A -85,B 0,C 180,E1 18482.228,E2 18482.228} C_VEL
LIN {X 0,Y 401.862,Z 412.544,A -85,B 0,C 180,E1 18481.634,E2 18481.634} C_VEL
LIN {X 0,Y 400.234,Z 430.959,A -85,B 0,C 180,E1 18480.804,E2 18480.804} C_VEL
LIN {X 0,Y 398.137,Z 448.72,A -85,B 0,C 180,E1 18479.734,E2 18479.734} C_VEL
LIN {X 0,Y 395.587,Z 466.297,A -85,B 0,C 180,E1 18478.37,E2 18478.37} C_VEL
LIN {X 0,Y 392.951,Z 482.019,A -85,B 0,C 180,E1 18476.848,E2 18476.848} C_VEL
LIN {X 0,Y 390.077,Z 497.356,A -85,B 0,C 180,E1 18475.019,E2 18475.019} C_VEL
LIN {X 0,Y 387.404,Z 510.623,A -85,B 0,C 180,E1 18473.096,E2 18473.096} C_VEL
LIN {X 0,Y 384.731,Z 523.341,A -85,B 0,C 180,E1 18470.856,E2 18470.856} C_VEL
LIN {X 0,Y 382.348,Z 534.532,A -85,B 0,C 180,E1 18468.445,E2 18468.445} C_VEL
LIN {X 0,Y 380.292,Z 544.495,A -85,B 0,C 180,E1 18465.785,E2 18465.785} C_VEL
LIN {X 0,Y 379.297,Z 549.518,A -85,B 0,C 180,E1 18464.165,E2 18464.165} C_VEL
LIN {X 0,Y 377.752,Z 552.648,A -85,B 0,C 180,E1 18463.108,E2 18463.108} C_VEL
LIN {X 0,Y 370.571,Z 559.827,A -85,B 0,C 180,E1 18460.345,E2 18460.345} C_VEL
LIN {X 0,Y 369.403,Z 561.837,A -85,B 0,C 180,E1 18459.29,E2 18459.29} C_VEL
LIN {X 0,Y 368.789,Z 566.125,A -85,B 0,C 180,E1 18456.225,E2 18456.225} C_VEL
LIN {X 0,Y 368.494,Z 568.703,A -85,B 0,C 180,E1 18453.11,E2 18453.11} C_VEL
LIN {X 0,Y 368.419,Z 569.569,A -85,B 0,C 180,E1 18449.999,E2 18449.999} C_VEL
LIN {X 0,Y 368.49,Z 568.761,A -85,B 0,C 180,E1 18446.888,E2 18446.888} C_VEL
LIN {X 0,Y 368.78,Z 566.245,A -85,B 0,C 180,E1 18443.773,E2 18443.773} C_VEL
LIN {X 0,Y 369.397,Z 561.913,A -85,B 0,C 180,E1 18440.653,E2 18440.653} C_VEL
LIN {X 0,Y 370.408,Z 556.003,A -85,B 0,C 180,E1 18437.686,E2 18437.686} C_VEL
LIN {X 0,Y 371.89,Z 548.497,A -85,B 0,C 180,E1 18434.842,E2 18434.842} C_VEL
LIN {X 0,Y 373.869,Z 539.22,A -85,B 0,C 180,E1 18432.087,E2 18432.087} C_VEL
LIN {X 0,Y 376.17,Z 528.925,A -85,B 0,C 180,E1 18429.622,E2 18429.622} C_VEL
LIN {X 0,Y 378.789,Z 517.255,A -85,B 0,C 180,E1 18427.331,E2 18427.331} C_VEL
LIN {X 0,Y 381.691,Z 503.88,A -85,B 0,C 180,E1 18425.178,E2 18425.178} C_VEL
LIN {X 0,Y 384.72,Z 489.01,A -85,B 0,C 180,E1 18423.221,E2 18423.221} C_VEL
LIN {X 0,Y 387.552,Z 473.716,A -85,B 0,C 180,E1 18421.575,E2 18421.575} C_VEL
LIN {X 0,Y 390.289,Z 456.868,A -85,B 0,C 180,E1 18420.113,E2 18420.113} C_VEL
LIN {X 0,Y 392.59,Z 440.019,A -85,B 0,C 180,E1 18418.953,E2 18418.953} C_VEL
LIN {X 0,Y 394.613,Z 421.124,A -85,B 0,C 180,E1 18417.959,E2 18417.959} C_VEL
LIN {X 0,Y 396.058,Z 401.976,A -85,B 0,C 180,E1 18417.245,E2 18417.245} C_VEL
LIN {X 0,Y 396.898,Z 381.943,A -85,B 0,C 180,E1 18416.778,E2 18416.778} C_VEL
LIN {X 0,Y 401.216,Z 212.447,A -85,B 0,C 180,E1 18413.792,E2 18413.792} C_VEL
LIN {X 0,Y 396.733,Z 185.304,A -85,B 0,C 180,E1 18412.668,E2 18412.668} C_VEL
LIN {X 0,Y 389.706,Z 172.485,A -85,B 0,C 180,E1 18411.493,E2 18411.493} C_VEL
LIN {X 0,Y 383.821,Z 156.243,A -85,B 0,C 180,E1 18408.499,E2 18408.499} C_VEL
LIN {X 0,Y 378.007,Z 142.164,A -85,B 0,C 180,E1 18405.576,E2 18405.576} C_VEL
LIN {X 0,Y 373.192,Z 131.313,A -85,B 0,C 180,E1 18403.095,E2 18403.095} C_VEL
LIN {X 0,Y 371.504,Z 128.325,A -85,B 0,C 180,E1 18402.308,E2 18402.308} C_VEL
LIN {X 0,Y 379.597,Z 148.64,A -85,B 0,C 180,E1 18399.405,E2 18399.405} C_VEL
LIN {X 0,Y 387.55,Z 171.256,A -85,B 0,C 180,E1 18396.394,E2 18396.394} C_VEL
LIN {X 0,Y 388.716,Z 175.424,A -85,B 0,C 180,E1 18395.879,E2 18395.879} C_VEL
LIN {X 0,Y 388.15,Z 187.437,A -85,B 0,C 180,E1 18394.797,E2 18394.797} C_VEL
LIN {X 0,Y 390.854,Z 210.314,A -85,B 0,C 180,E1 18393.955,E2 18393.955} C_VEL
LIN {X 0,Y 383.397,Z 399.191,A -85,B 0,C 180,E1 18389.526,E2 18389.526} C_VEL
LIN {X 0,Y 382.422,Z 418.391,A -85,B 0,C 180,E1 18388.799,E2 18388.799} C_VEL
LIN {X 0,Y 381.17,Z 436.84,A -85,B 0,C 180,E1 18387.835,E2 18387.835} C_VEL
LIN {X 0,Y 379.646,Z 455.079,A -85,B 0,C 180,E1 18386.598,E2 18386.598} C_VEL
LIN {X 0,Y 377.905,Z 473.232,A -85,B 0,C 180,E1 18385.045,E2 18385.045} C_VEL
LIN {X 0,Y 376.187,Z 489.488,A -85,B 0,C 180,E1 18383.33,E2 18383.33} C_VEL
LIN {X 0,Y 374.476,Z 504.752,A -85,B 0,C 180,E1 18381.375,E2 18381.375} C_VEL
LIN {X 0,Y 372.91,Z 518.372,A -85,B 0,C 180,E1 18379.257,E2 18379.257} C_VEL
LIN {X 0,Y 371.494,Z 530.852,A -85,B 0,C 180,E1 18376.899,E2 18376.899} C_VEL
LIN {X 0,Y 370.408,Z 541.136,A -85,B 0,C 180,E1 18374.539,E2 18374.539} C_VEL
LIN {X 0,Y 369.564,Z 550.048,A -85,B 0,C 180,E1 18372.024,E2 18372.024} C_VEL
LIN {X 0,Y 368.973,Z 557.509,A -85,B 0,C 180,E1 18369.358,E2 18369.358} C_VEL
LIN {X 0,Y 368.633,Z 563.139,A -85,B 0,C 180,E1 18366.698,E2 18366.698} C_VEL
LIN {X 0,Y 368.469,Z 567.27,A -85,B 0,C 180,E1 18363.89,E2 18363.89} C_VEL
LIN {X 0,Y 368.437,Z 569.532,A -85,B 0,C 180,E1 18361.244,E2 18361.244} C_VEL
LIN {X 0,Y 368.501,Z 570.248,A -85,B 0,C 180,E1 18358.601,E2 18358.601} C_VEL
LIN {X 0,Y 368.686,Z 569.328,A -85,B 0,C 180,E1 18355.801,E2 18355.801} C_VEL
LIN {X 0,Y 369.047,Z 566.668,A -85,B 0,C 180,E1 18352.997,E2 18352.997} C_VEL
LIN {X 0,Y 369.616,Z 562.47,A -85,B 0,C 180,E1 18350.345,E2 18350.345} C_VEL
LIN {X 0,Y 370.506,Z 556.501,A -85,B 0,C 180,E1 18347.665,E2 18347.665} C_VEL
LIN {X 0,Y 371.741,Z 548.731,A -85,B 0,C 180,E1 18345.037,E2 18345.037} C_VEL
LIN {X 0,Y 373.293,Z 539.386,A -85,B 0,C 180,E1 18342.543,E2 18342.543} C_VEL
LIN {X 0,Y 375.098,Z 528.492,A -85,B 0,C 180,E1 18340.213,E2 18340.213} C_VEL
LIN {X 0,Y 377.198,Z 515.671,A -85,B 0,C 180,E1 18337.971,E2 18337.971} C_VEL
LIN {X 0,Y 379.464,Z 501.112,A -85,B 0,C 180,E1 18335.895,E2 18335.895} C_VEL
LIN {X 0,Y 381.646,Z 486.123,A -85,B 0,C 180,E1 18334.138,E2 18334.138} C_VEL
LIN {X 0,Y 383.844,Z 469.579,A -85,B 0,C 180,E1 18332.545,E2 18332.545} C_VEL
LIN {X 0,Y 385.87,Z 451.979,A -85,B 0,C 180,E1 18331.187,E2 18331.187} C_VEL
LIN {X 0,Y 387.682,Z 433.731,A -85,B 0,C 180,E1 18330.063,E2 18330.063} C_VEL
LIN {X 0,Y 389.414,Z 412.37,A -85,B 0,C 180,E1 18329.072,E2 18329.072} C_VEL
LIN {X 0,Y 391.801,Z 377.99,A -85,B 0,C 180,E1 18327.989,E2 18327.989} C_VEL
LIN {X 0,Y 398.485,Z 307.609,A -85,B 0,C 180,E1 18325.808,E2 18325.808} C_VEL
LIN {X 0,Y 408.874,Z 224.092,A -85,B 0,C 180,E1 18323.122,E2 18323.122} C_VEL
LIN {X 0,Y 409.975,Z 215.563,A -85,B 0,C 180,E1 18322.817,E2 18322.817} C_VEL
LIN {X 0,Y 410.14,Z 205.576,A -85,B 0,C 180,E1 18322.008,E2 18322.008} C_VEL
LIN {X 0,Y 412.572,Z 191.432,A -85,B 0,C 180,E1 18320.584,E2 18320.584} C_VEL
LIN {X 0,Y 411.997,Z 185.315,A -85,B 0,C 180,E1 18319.062,E2 18319.062} C_VEL
LIN {X 0,Y 411.58,Z 181.237,A -85,B 0,C 180,E1 18317.606,E2 18317.606} C_VEL
LIN {X 0,Y 411.509,Z 179.169,A -85,B 0,C 180,E1 18316.559,E2 18316.559} C_VEL
LIN {X 0,Y 411.405,Z 178.765,A -85,B 0,C 180,E1 18315.804,E2 18315.804} C_VEL
LIN {X 0,Y 409.672,Z 184.687,A -85,B 0,C 180,E1 18314.269,E2 18314.269} C_VEL
LIN {X 0,Y 408.92,Z 190.413,A -85,B 0,C 180,E1 18313.016,E2 18313.016} C_VEL
LIN {X 0,Y 408.8,Z 191.491,A -85,B 0,C 180,E1 18312.84,E2 18312.84} C_VEL
LIN {X 0,Y 406.674,Z 201.169,A -85,B 0,C 180,E1 18312.197,E2 18312.197} C_VEL
LIN {X 0,Y 402.956,Z 216.762,A -85,B 0,C 180,E1 18311.564,E2 18311.564} C_VEL
LIN {X 0,Y 395.54,Z 418.334,A -85,B 0,C 180,E1 18307.533,E2 18307.533} C_VEL
LIN {X 0,Y 393.806,Z 440.152,A -85,B 0,C 180,E1 18306.844,E2 18306.844} C_VEL
LIN {X 0,Y 391.541,Z 461.439,A -85,B 0,C 180,E1 18305.879,E2 18305.879} C_VEL
LIN {X 0,Y 388.981,Z 481.116,A -85,B 0,C 180,E1 18304.697,E2 18304.697} C_VEL
LIN {X 0,Y 386.123,Z 500.361,A -85,B 0,C 180,E1 18303.238,E2 18303.238} C_VEL
LIN {X 0,Y 383.167,Z 518.489,A -85,B 0,C 180,E1 18301.548,E2 18301.548} C_VEL
LIN {X 0,Y 380.257,Z 535.519,A -85,B 0,C 180,E1 18299.627,E2 18299.627} C_VEL
LIN {X 0,Y 377.402,Z 551.744,A -85,B 0,C 180,E1 18297.437,E2 18297.437} C_VEL
LIN {X 0,Y 374.739,Z 567.218,A -85,B 0,C 180,E1 18294.934,E2 18294.934} C_VEL
LIN {X 0,Y 372.59,Z 580.365,A -85,B 0,C 180,E1 18292.4,E2 18292.4} C_VEL
LIN {X 0,Y 370.861,Z 592.158,A -85,B 0,C 180,E1 18289.695,E2 18289.695} C_VEL
LIN {X 0,Y 369.57,Z 602.537,A -85,B 0,C 180,E1 18286.828,E2 18286.828} C_VEL
LIN {X 0,Y 368.714,Z 611.374,A -85,B 0,C 180,E1 18283.807,E2 18283.807} C_VEL
LIN {X 0,Y 368.289,Z 618.3,A -85,B 0,C 180,E1 18280.798,E2 18280.798} C_VEL
LIN {X 0,Y 368.148,Z 623.469,A -85,B 0,C 180,E1 18277.806,E2 18277.806} C_VEL
LIN {X 0,Y 368.154,Z 626.974,A -85,B 0,C 180,E1 18274.831,E2 18274.831} C_VEL
LIN {X 0,Y 368.199,Z 628.759,A -85,B 0,C 180,E1 18272.024,E2 18272.024} C_VEL
LIN {X 0,Y 368.217,Z 629.056,A -85,B 0,C 180,E1 18269.223,E2 18269.223} C_VEL
LIN {X 0,Y 368.173,Z 627.842,A -85,B 0,C 180,E1 18266.264,E2 18266.264} C_VEL
LIN {X 0,Y 368.135,Z 625.16,A -85,B 0,C 180,E1 18263.451,E2 18263.451} C_VEL
LIN {X 0,Y 368.207,Z 620.684,A -85,B 0,C 180,E1 18260.466,E2 18260.466} C_VEL
LIN {X 0,Y 368.487,Z 614.494,A -85,B 0,C 180,E1 18257.464,E2 18257.464} C_VEL
LIN {X 0,Y 369.107,Z 606.96,A -85,B 0,C 180,E1 18254.606,E2 18254.606} C_VEL
LIN {X 0,Y 370.217,Z 597.026,A -85,B 0,C 180,E1 18251.581,E2 18251.581} C_VEL
LIN {X 0,Y 371.812,Z 585.493,A -85,B 0,C 180,E1 18248.714,E2 18248.714} C_VEL
LIN {X 0,Y 373.872,Z 572.42,A -85,B 0,C 180,E1 18246.016,E2 18246.016} C_VEL
LIN {X 0,Y 376.249,Z 558.344,A -85,B 0,C 180,E1 18243.579,E2 18243.579} C_VEL
LIN {X 0,Y 378.976,Z 542.729,A -85,B 0,C 180,E1 18241.305,E2 18241.305} C_VEL
LIN {X 0,Y 381.945,Z 525.595,A -85,B 0,C 180,E1 18239.219,E2 18239.219} C_VEL
LIN {X 0,Y 384.974,Z 507.42,A -85,B 0,C 180,E1 18237.391,E2 18237.391} C_VEL
LIN {X 0,Y 387.92,Z 488.202,A -85,B 0,C 180,E1 18235.815,E2 18235.815} C_VEL
LIN {X 0,Y 390.533,Z 469.111,A -85,B 0,C 180,E1 18234.558,E2 18234.558} C_VEL
LIN {X 0,Y 392.873,Z 449.25,A -85,B 0,C 180,E1 18233.542,E2 18233.542} C_VEL
LIN {X 0,Y 394.783,Z 428.619,A -85,B 0,C 180,E1 18232.764,E2 18232.764} C_VEL
LIN {X 0,Y 396.057,Z 406.511,A -85,B 0,C 180,E1 18232.207,E2 18232.207} C_VEL
LIN {X 0,Y 403.487,Z 199.036,A -85,B 0,C 180,E1 18228.102,E2 18228.102} C_VEL
LIN {X 0,Y 402.196,Z 189.219,A -85,B 0,C 180,E1 18227.722,E2 18227.722} C_VEL
LIN {X 0,Y 391.046,Z 169.41,A -85,B 0,C 180,E1 18225.876,E2 18225.876} C_VEL
LIN {X 0,Y 388.661,Z 165.205,A -85,B 0,C 180,E1 18225.447,E2 18225.447} C_VEL
LIN {X 0,Y 381.379,Z 148.111,A -85,B 0,C 180,E1 18222.328,E2 18222.328} C_VEL
LIN {X 0,Y 375.403,Z 135.48,A -85,B 0,C 180,E1 18219.734,E2 18219.734} C_VEL
LIN {X 0,Y 371.522,Z 127.502,A -85,B 0,C 180,E1 18217.953,E2 18217.953} C_VEL
LIN {X 0,Y 369.83,Z 124.177,A -85,B 0,C 180,E1 18217.165,E2 18217.165} C_VEL
LIN {X 0,Y 369.691,Z 123.376,A -85,B 0,C 180,E1 18216.976,E2 18216.976} C_VEL
LIN {X 0,Y 369.698,Z 123.413,A -85,B 0,C 180,E1 18212.929,E2 18212.929} C_VEL
LIN {X 0,Y 369.697,Z 123.413,A -85,B 0,C 180,E1 18208.954,E2 18208.954} C_VEL
LIN {X 0,Y 369.696,Z 123.417,A -85,B 0,C 180,E1 18204.955,E2 18204.955} C_VEL
LIN {X 0,Y 369.7,Z 123.433,A -85,B 0,C 180,E1 18200.915,E2 18200.915} C_VEL
LIN {X 0,Y 369.704,Z 123.428,A -85,B 0,C 180,E1 18196.821,E2 18196.821} C_VEL
LIN {X 0,Y 369.701,Z 123.403,A -85,B 0,C 180,E1 18192.813,E2 18192.813} C_VEL
LIN {X 0,Y 369.709,Z 123.416,A -85,B 0,C 180,E1 18188.711,E2 18188.711} C_VEL
LIN {X 0,Y 369.715,Z 123.429,A -85,B 0,C 180,E1 18184.653,E2 18184.653} C_VEL
LIN {X 0,Y 369.73,Z 123.398,A -85,B 0,C 180,E1 18180.465,E2 18180.465} C_VEL
LIN {X 0,Y 369.714,Z 123.418,A -85,B 0,C 180,E1 18176.29,E2 18176.29} C_VEL
LIN {X 0,Y 369.713,Z 123.428,A -85,B 0,C 180,E1 18172.228,E2 18172.228} C_VEL
LIN {X 0,Y 369.7,Z 123.403,A -85,B 0,C 180,E1 18168.138,E2 18168.138} C_VEL
LIN {X 0,Y 369.7,Z 123.424,A -85,B 0,C 180,E1 18164.147,E2 18164.147} C_VEL
LIN {X 0,Y 369.695,Z 123.432,A -85,B 0,C 180,E1 18160.076,E2 18160.076} C_VEL
LIN {X 0,Y 369.688,Z 123.409,A -85,B 0,C 180,E1 18156.065,E2 18156.065} C_VEL
LIN {X 0,Y 369.688,Z 123.408,A -85,B 0,C 180,E1 18152.102,E2 18152.102} C_VEL
LIN {X 0,Y 369.69,Z 123.423,A -85,B 0,C 180,E1 18148.127,E2 18148.127} C_VEL
LIN {X 0,Y 369.683,Z 123.431,A -85,B 0,C 180,E1 18144.062,E2 18144.062} C_VEL
LIN {X 0,Y 369.685,Z 123.43,A -85,B 0,C 180,E1 18140.133,E2 18140.133} C_VEL
LIN {X 0,Y 369.742,Z 123.593,A -85,B 0,C 180,E1 18138.663,E2 18138.663} C_VEL
LIN {X 0,Y 371.051,Z 127.017,A -85,B 0,C 180,E1 18137.857,E2 18137.857} C_VEL
LIN {X 0,Y 373.897,Z 133.107,A -85,B 0,C 180,E1 18136.375,E2 18136.375} C_VEL
LIN {X 0,Y 379.458,Z 145.615,A -85,B 0,C 180,E1 18133.563,E2 18133.563} C_VEL
LIN {X 0,Y 385.264,Z 160.15,A -85,B 0,C 180,E1 18130.646,E2 18130.646} C_VEL
LIN {X 0,Y 389.967,Z 173.06,A -85,B 0,C 180,E1 18128.345,E2 18128.345} C_VEL
LIN {X 0,Y 396.956,Z 186.101,A -85,B 0,C 180,E1 18127.177,E2 18127.177} C_VEL
LIN {X 0,Y 401.249,Z 214.143,A -85,B 0,C 180,E1 18126.061,E2 18126.061} C_VEL
LIN {X 0,Y 396.461,Z 393.565,A -85,B 0,C 180,E1 18122.883,E2 18122.883} C_VEL
LIN {X 0,Y 395.248,Z 412.927,A -85,B 0,C 180,E1 18122.28,E2 18122.28} C_VEL
LIN {X 0,Y 393.604,Z 430.851,A -85,B 0,C 180,E1 18121.467,E2 18121.467} C_VEL
LIN {X 0,Y 391.414,Z 448.725,A -85,B 0,C 180,E1 18120.382,E2 18120.382} C_VEL
LIN {X 0,Y 388.806,Z 466.053,A -85,B 0,C 180,E1 18119.031,E2 18119.031} C_VEL
LIN {X 0,Y 385.988,Z 482.188,A -85,B 0,C 180,E1 18117.456,E2 18117.456} C_VEL
LIN {X 0,Y 383.09,Z 497.038,A -85,B 0,C 180,E1 18115.673,E2 18115.673} C_VEL
LIN {X 0,Y 380.058,Z 511.367,A -85,B 0,C 180,E1 18113.57,E2 18113.57} C_VEL
LIN {X 0,Y 377.253,Z 524.055,A -85,B 0,C 180,E1 18111.29,E2 18111.29} C_VEL
LIN {X 0,Y 374.746,Z 535.226,A -85,B 0,C 180,E1 18108.834,E2 18108.834} C_VEL
LIN {X 0,Y 372.555,Z 545.254,A -85,B 0,C 180,E1 18106.095,E2 18106.095} C_VEL
LIN {X 0,Y 370.87,Z 553.491,A -85,B 0,C 180,E1 18103.246,E2 18103.246} C_VEL
LIN {X 0,Y 369.732,Z 559.764,A -85,B 0,C 180,E1 18100.438,E2 18100.438} C_VEL
LIN {X 0,Y 369.403,Z 561.837,A -85,B 0,C 180,E1 18099.29,E2 18099.29} C_VEL
LIN {X 0,Y 368.141,Z 563.848,A -85,B 0,C 180,E1 18098.142,E2 18098.142} C_VEL
LIN {X 0,Y 363.153,Z 567.004,A -85,B 0,C 180,E1 18095.959,E2 18095.959} C_VEL
LIN {X 0,Y 360.826,Z 568.457,A -85,B 0,C 180,E1 18094.517,E2 18094.517} C_VEL
LIN {X 0,Y 360.577,Z 568.816,A -85,B 0,C 180,E1 18093.99,E2 18093.99} C_VEL
LIN {X 0,Y 360.446,Z 570.109,A -85,B 0,C 180,E1 18090.794,E2 18090.794} C_VEL
LIN {X 0,Y 360.484,Z 569.719,A -85,B 0,C 180,E1 18087.615,E2 18087.615} C_VEL
LIN {X 0,Y 360.724,Z 567.638,A -85,B 0,C 180,E1 18084.432,E2 18084.432} C_VEL
LIN {X 0,Y 361.284,Z 563.786,A -85,B 0,C 180,E1 18081.244,E2 18081.244} C_VEL
LIN {X 0,Y 362.23,Z 558.363,A -85,B 0,C 180,E1 18078.213,E2 18078.213} C_VEL
LIN {X 0,Y 363.725,Z 551.055,A -85,B 0,C 180,E1 18075.187,E2 18075.187} C_VEL
LIN {X 0,Y 365.587,Z 542.697,A -85,B 0,C 180,E1 18072.491,E2 18072.491} C_VEL
LIN {X 0,Y 368.004,Z 532.35,A -85,B 0,C 180,E1 18069.814,E2 18069.814} C_VEL
LIN {X 0,Y 370.821,Z 520.434,A -85,B 0,C 180,E1 18067.32,E2 18067.32} C_VEL
LIN {X 0,Y 373.71,Z 507.846,A -85,B 0,C 180,E1 18065.161,E2 18065.161} C_VEL
LIN {X 0,Y 376.885,Z 493.238,A -85,B 0,C 180,E1 18063.106,E2 18063.106} C_VEL
LIN {X 0,Y 379.883,Z 478.181,A -85,B 0,C 180,E1 18061.377,E2 18061.377} C_VEL
LIN {X 0,Y 382.778,Z 461.667,A -85,B 0,C 180,E1 18059.839,E2 18059.839} C_VEL
LIN {X 0,Y 385.353,Z 444.444,A -85,B 0,C 180,E1 18058.564,E2 18058.564} C_VEL
LIN {X 0,Y 387.489,Z 426.531,A -85,B 0,C 180,E1 18057.539,E2 18057.539} C_VEL
LIN {X 0,Y 389.179,Z 407.36,A -85,B 0,C 180,E1 18056.74,E2 18056.74} C_VEL
LIN {X 0,Y 390.227,Z 387.772,A -85,B 0,C 180,E1 18056.205,E2 18056.205} C_VEL
LIN {X 0,Y 394.984,Z 213.811,A -85,B 0,C 180,E1 18053.085,E2 18053.085} C_VEL
LIN {X 0,Y 390.947,Z 189.032,A -85,B 0,C 180,E1 18052.033,E2 18052.033} C_VEL
LIN {X 0,Y 381.634,Z 172.089,A -85,B 0,C 180,E1 18050.378,E2 18050.378} C_VEL
LIN {X 0,Y 375.998,Z 156.943,A -85,B 0,C 180,E1 18047.443,E2 18047.443} C_VEL
LIN {X 0,Y 370.134,Z 142.995,A -85,B 0,C 180,E1 18044.399,E2 18044.399} C_VEL
LIN {X 0,Y 366.384,Z 134.859,A -85,B 0,C 180,E1 18042.435,E2 18042.435} C_VEL
LIN {X 0,Y 365.878,Z 134.635,A -85,B 0,C 180,E1 18042.262,E2 18042.262} C_VEL
LIN {X 0,Y 374.134,Z 156.069,A -85,B 0,C 180,E1 18039.193,E2 18039.193} C_VEL
LIN {X 0,Y 381.551,Z 177.642,A -85,B 0,C 180,E1 18036.316,E2 18036.316} C_VEL
LIN {X 0,Y 381.089,Z 187.903,A -85,B 0,C 180,E1 18035.386,E2 18035.386} C_VEL
LIN {X 0,Y 383.788,Z 211.393,A -85,B 0,C 180,E1 18034.5,E2 18034.5} C_VEL
LIN {X 0,Y 375.96,Z 399.8,A -85,B 0,C 180,E1 18029.963,E2 18029.963} C_VEL
LIN {X 0,Y 374.929,Z 419.166,A -85,B 0,C 180,E1 18029.211,E2 18029.211} C_VEL
LIN {X 0,Y 373.54,Z 438.636,A -85,B 0,C 180,E1 18028.16,E2 18028.16} C_VEL
LIN {X 0,Y 371.912,Z 457.252,A -85,B 0,C 180,E1 18026.85,E2 18026.85} C_VEL
LIN {X 0,Y 370.207,Z 474.313,A -85,B 0,C 180,E1 18025.346,E2 18025.346} C_VEL
LIN {X 0,Y 368.43,Z 490.512,A -85,B 0,C 180,E1 18023.597,E2 18023.597} C_VEL
LIN {X 0,Y 366.637,Z 505.919,A -85,B 0,C 180,E1 18021.572,E2 18021.572} C_VEL
LIN {X 0,Y 364.985,Z 519.737,A -85,B 0,C 180,E1 18019.359,E2 18019.359} C_VEL
LIN {X 0,Y 363.625,Z 531.388,A -85,B 0,C 180,E1 18017.111,E2 18017.111} C_VEL
LIN {X 0,Y 362.495,Z 541.722,A -85,B 0,C 180,E1 18014.701,E2 18014.701} C_VEL
LIN {X 0,Y 361.619,Z 550.679,A -85,B 0,C 180,E1 18012.131,E2 18012.131} C_VEL
LIN {X 0,Y 361.006,Z 558.183,A -85,B 0,C 180,E1 18009.405,E2 18009.405} C_VEL
LIN {X 0,Y 360.655,Z 563.845,A -85,B 0,C 180,E1 18006.687,E2 18006.687} C_VEL
LIN {X 0,Y 360.495,Z 567.808,A -85,B 0,C 180,E1 18003.976,E2 18003.976} C_VEL
LIN {X 0,Y 360.466,Z 570.256,A -85,B 0,C 180,E1 18001.113,E2 18001.113} C_VEL
LIN {X 0,Y 360.542,Z 570.974,A -85,B 0,C 180,E1 17998.411,E2 17998.411} C_VEL
LIN {X 0,Y 360.754,Z 570.054,A -85,B 0,C 180,E1 17995.549,E2 17995.549} C_VEL
LIN {X 0,Y 361.169,Z 567.381,A -85,B 0,C 180,E1 17992.684,E2 17992.684} C_VEL
LIN {X 0,Y 361.814,Z 563.19,A -85,B 0,C 180,E1 17989.974,E2 17989.974} C_VEL
LIN {X 0,Y 362.788,Z 557.241,A -85,B 0,C 180,E1 17987.263,E2 17987.263} C_VEL
LIN {X 0,Y 364.171,Z 549.422,A -85,B 0,C 180,E1 17984.555,E2 17984.555} C_VEL
LIN {X 0,Y 365.878,Z 539.923,A -85,B 0,C 180,E1 17981.992,E2 17981.992} C_VEL
LIN {X 0,Y 367.839,Z 529.146,A -85,B 0,C 180,E1 17979.64,E2 17979.64} C_VEL
LIN {X 0,Y 370.098,Z 516.344,A -85,B 0,C 180,E1 17977.367,E2 17977.367} C_VEL
LIN {X 0,Y 372.462,Z 502.347,A -85,B 0,C 180,E1 17975.328,E2 17975.328} C_VEL
LIN {X 0,Y 374.923,Z 486.864,A -85,B 0,C 180,E1 17973.468,E2 17973.468} C_VEL
LIN {X 0,Y 377.404,Z 469.498,A -85,B 0,C 180,E1 17971.778,E2 17971.778} C_VEL
LIN {X 0,Y 379.601,Z 451.923,A -85,B 0,C 180,E1 17970.405,E2 17970.405} C_VEL
LIN {X 0,Y 381.709,Z 432.578,A -85,B 0,C 180,E1 17969.205,E2 17969.205} C_VEL
LIN {X 0,Y 383.476,Z 412.295,A -85,B 0,C 180,E1 17968.262,E2 17968.262} C_VEL
LIN {X 0,Y 387.086,Z 368.915,A -85,B 0,C 180,E1 17966.853,E2 17966.853} C_VEL
LIN {X 0,Y 394.985,Z 297.75,A -85,B 0,C 180,E1 17964.538,E2 17964.538} C_VEL
LIN {X 0,Y 406.213,Z 218.157,A -85,B 0,C 180,E1 17961.888,E2 17961.888} C_VEL
LIN {X 0,Y 406.674,Z 207.401,A -85,B 0,C 180,E1 17960.981,E2 17960.981} C_VEL
LIN {X 0,Y 408.851,Z 196.612,A -85,B 0,C 180,E1 17959.88,E2 17959.88} C_VEL
LIN {X 0,Y 408.619,Z 191.042,A -85,B 0,C 180,E1 17958.369,E2 17958.369} C_VEL
LIN {X 0,Y 408.623,Z 187.797,A -85,B 0,C 180,E1 17957.024,E2 17957.024} C_VEL
LIN {X 0,Y 408.722,Z 186.422,A -85,B 0,C 180,E1 17956.188,E2 17956.188} C_VEL
LIN {X 0,Y 408.519,Z 186.882,A -85,B 0,C 180,E1 17955.965,E2 17955.965} C_VEL
LIN {X 0,Y 406.794,Z 192.435,A -85,B 0,C 180,E1 17954.538,E2 17954.538} C_VEL
LIN {X 0,Y 406.289,Z 195.874,A -85,B 0,C 180,E1 17953.752,E2 17953.752} C_VEL
LIN {X 0,Y 404.305,Z 203.485,A -85,B 0,C 180,E1 17953.239,E2 17953.239} C_VEL
LIN {X 0,Y 399.38,Z 222.469,A -85,B 0,C 180,E1 17952.493,E2 17952.493} C_VEL
LIN {X 0,Y 395.661,Z 243.707,A -85,B 0,C 180,E1 17951.748,E2 17951.748} C_VEL
LIN {X 0,Y 389.012,Z 417.888,A -85,B 0,C 180,E1 17948.217,E2 17948.217} C_VEL
LIN {X 0,Y 387.22,Z 439.682,A -85,B 0,C 180,E1 17947.523,E2 17947.523} C_VEL
LIN {X 0,Y 384.877,Z 460.785,A -85,B 0,C 180,E1 17946.558,E2 17946.558} C_VEL
LIN {X 0,Y 382.136,Z 481.017,A -85,B 0,C 180,E1 17945.328,E2 17945.328} C_VEL
LIN {X 0,Y 379.079,Z 500.615,A -85,B 0,C 180,E1 17943.815,E2 17943.815} C_VEL
LIN {X 0,Y 376.038,Z 518.333,A -85,B 0,C 180,E1 17942.127,E2 17942.127} C_VEL
LIN {X 0,Y 372.975,Z 535.297,A -85,B 0,C 180,E1 17940.176,E2 17940.176} C_VEL
LIN {X 0,Y 369.982,Z 551.43,A -85,B 0,C 180,E1 17937.954,E2 17937.954} C_VEL
LIN {X 0,Y 367.239,Z 566.446,A -85,B 0,C 180,E1 17935.48,E2 17935.48} C_VEL
LIN {X 0,Y 364.944,Z 579.62,A -85,B 0,C 180,E1 17932.896,E2 17932.896} C_VEL
LIN {X 0,Y 363.075,Z 591.548,A -85,B 0,C 180,E1 17930.105,E2 17930.105} C_VEL
LIN {X 0,Y 361.638,Z 602.336,A -85,B 0,C 180,E1 17927.043,E2 17927.043} C_VEL
LIN {X 0,Y 360.741,Z 611.117,A -85,B 0,C 180,E1 17923.955,E2 17923.955} C_VEL
LIN {X 0,Y 360.297,Z 617.953,A -85,B 0,C 180,E1 17920.878,E2 17920.878} C_VEL
LIN {X 0,Y 360.159,Z 623.034,A -85,B 0,C 180,E1 17917.819,E2 17917.819} C_VEL
LIN {X 0,Y 360.175,Z 626.485,A -85,B 0,C 180,E1 17914.732,E2 17914.732} C_VEL
LIN {X 0,Y 360.226,Z 628.252,A -85,B 0,C 180,E1 17911.751,E2 17911.751} C_VEL
LIN {X 0,Y 360.243,Z 628.361,A -85,B 0,C 180,E1 17908.888,E2 17908.888} C_VEL
LIN {X 0,Y 360.187,Z 626.944,A -85,B 0,C 180,E1 17905.862,E2 17905.862} C_VEL
LIN {X 0,Y 360.153,Z 624.145,A -85,B 0,C 180,E1 17902.985,E2 17902.985} C_VEL
LIN {X 0,Y 360.237,Z 619.462,A -85,B 0,C 180,E1 17899.931,E2 17899.931} C_VEL
LIN {X 0,Y 360.586,Z 613.047,A -85,B 0,C 180,E1 17896.859,E2 17896.859} C_VEL
LIN {X 0,Y 361.352,Z 604.772,A -85,B 0,C 180,E1 17893.769,E2 17893.769} C_VEL
LIN {X 0,Y 362.558,Z 595.082,A -85,B 0,C 180,E1 17890.843,E2 17890.843} C_VEL
LIN {X 0,Y 364.222,Z 584.044,A -85,B 0,C 180,E1 17888.079,E2 17888.079} C_VEL
LIN {X 0,Y 366.49,Z 570.682,A -85,B 0,C 180,E1 17885.297,E2 17885.297} C_VEL
LIN {X 0,Y 369.277,Z 555.277,A -85,B 0,C 180,E1 17882.635,E2 17882.635} C_VEL
LIN {X 0,Y 372.337,Z 538.826,A -85,B 0,C 180,E1 17880.275,E2 17880.275} C_VEL
LIN {X 0,Y 375.508,Z 521.256,A -85,B 0,C 180,E1 17878.184,E2 17878.184} C_VEL
LIN {X 0,Y 378.66,Z 503.033,A -85,B 0,C 180,E1 17876.405,E2 17876.405} C_VEL
LIN {X 0,Y 381.633,Z 484.062,A -85,B 0,C 180,E1 17874.896,E2 17874.896} C_VEL
LIN {X 0,Y 384.248,Z 465.287,A -85,B 0,C 180,E1 17873.704,E2 17873.704} C_VEL
LIN {X 0,Y 386.65,Z 444.71,A -85,B 0,C 180,E1 17872.695,E2 17872.695} C_VEL
LIN {X 0,Y 388.587,Z 423.198,A -85,B 0,C 180,E1 17871.942,E2 17871.942} C_VEL
LIN {X 0,Y 389.928,Z 395.507,A -85,B 0,C 180,E1 17871.308,E2 17871.308} C_VEL
LIN {X 0,Y 397.236,Z 200.076,A -85,B 0,C 180,E1 17867.393,E2 17867.393} C_VEL
LIN {X 0,Y 396.291,Z 192.91,A -85,B 0,C 180,E1 17867.107,E2 17867.107} C_VEL
LIN {X 0,Y 385.674,Z 173.932,A -85,B 0,C 180,E1 17865.289,E2 17865.289} C_VEL
LIN {X 0,Y 380.535,Z 165.234,A -85,B 0,C 180,E1 17864.34,E2 17864.34} C_VEL
LIN {X 0,Y 373.828,Z 149.612,A -85,B 0,C 180,E1 17861.348,E2 17861.348} C_VEL
LIN {X 0,Y 367.96,Z 137.248,A -85,B 0,C 180,E1 17858.68,E2 17858.68} C_VEL
LIN {X 0,Y 365.215,Z 132.008,A -85,B 0,C 180,E1 17857.428,E2 17857.428} C_VEL
LIN {X 0,Y 363.484,Z 128.406,A -85,B 0,C 180,E1 17856.563,E2 17856.563} C_VEL
LIN {X 0,Y 362.006,Z 125.552,A -85,B 0,C 180,E1 17855.841,E2 17855.841} C_VEL
LIN {X 0,Y 361.761,Z 124.405,A -85,B 0,C 180,E1 17855.55,E2 17855.55} C_VEL
LIN {X 0,Y 361.76,Z 124.415,A -85,B 0,C 180,E1 17851.491,E2 17851.491} C_VEL
LIN {X 0,Y 361.758,Z 124.41,A -85,B 0,C 180,E1 17847.478,E2 17847.478} C_VEL
LIN {X 0,Y 361.753,Z 124.401,A -85,B 0,C 180,E1 17843.281,E2 17843.281} C_VEL
LIN {X 0,Y 361.752,Z 124.396,A -85,B 0,C 180,E1 17839.202,E2 17839.202} C_VEL
LIN {X 0,Y 361.754,Z 124.416,A -85,B 0,C 180,E1 17835.058,E2 17835.058} C_VEL
LIN {X 0,Y 361.756,Z 124.419,A -85,B 0,C 180,E1 17830.994,E2 17830.994} C_VEL
LIN {X 0,Y 361.753,Z 124.389,A -85,B 0,C 180,E1 17826.985,E2 17826.985} C_VEL
LIN {X 0,Y 361.764,Z 124.411,A -85,B 0,C 180,E1 17822.851,E2 17822.851} C_VEL
LIN {X 0,Y 361.761,Z 124.414,A -85,B 0,C 180,E1 17818.891,E2 17818.891} C_VEL
LIN {X 0,Y 361.767,Z 124.389,A -85,B 0,C 180,E1 17814.767,E2 17814.767} C_VEL
LIN {X 0,Y 361.772,Z 124.418,A -85,B 0,C 180,E1 17810.775,E2 17810.775} C_VEL
LIN {X 0,Y 361.785,Z 124.408,A -85,B 0,C 180,E1 17806.576,E2 17806.576} C_VEL
LIN {X 0,Y 361.776,Z 124.39,A -85,B 0,C 180,E1 17802.453,E2 17802.453} C_VEL
LIN {X 0,Y 361.765,Z 124.409,A -85,B 0,C 180,E1 17798.262,E2 17798.262} C_VEL
LIN {X 0,Y 361.756,Z 124.422,A -85,B 0,C 180,E1 17794.106,E2 17794.106} C_VEL
LIN {X 0,Y 361.751,Z 124.408,A -85,B 0,C 180,E1 17790.164,E2 17790.164} C_VEL
LIN {X 0,Y 361.755,Z 124.403,A -85,B 0,C 180,E1 17786.251,E2 17786.251} C_VEL
LIN {X 0,Y 361.747,Z 124.407,A -85,B 0,C 180,E1 17782.149,E2 17782.149} C_VEL
LIN {X 0,Y 361.766,Z 124.586,A -85,B 0,C 180,E1 17780.065,E2 17780.065} C_VEL
LIN {X 0,Y 363.075,Z 127.922,A -85,B 0,C 180,E1 17779.226,E2 17779.226} C_VEL
LIN {X 0,Y 364.003,Z 129.613,A -85,B 0,C 180,E1 17778.757,E2 17778.757} C_VEL
LIN {X 0,Y 369.626,Z 141.873,A -85,B 0,C 180,E1 17775.74,E2 17775.74} C_VEL
LIN {X 0,Y 375.479,Z 155.734,A -85,B 0,C 180,E1 17772.696,E2 17772.696} C_VEL
LIN {X 0,Y 381.624,Z 172.159,A -85,B 0,C 180,E1 17769.502,E2 17769.502} C_VEL
LIN {X 0,Y 391.162,Z 189.666,A -85,B 0,C 180,E1 17767.814,E2 17767.814} C_VEL
LIN {X 0,Y 395.006,Z 215.566,A -85,B 0,C 180,E1 17766.766,E2 17766.766} C_VEL
LIN {X 0,Y 389.959,Z 393.87,A -85,B 0,C 180,E1 17763.561,E2 17763.561} C_VEL
LIN {X 0,Y 388.696,Z 413.195,A -85,B 0,C 180,E1 17762.953,E2 17762.953} C_VEL
LIN {X 0,Y 386.949,Z 431.391,A -85,B 0,C 180,E1 17762.116,E2 17762.116} C_VEL
LIN {X 0,Y 384.589,Z 449.738,A -85,B 0,C 180,E1 17760.98,E2 17760.98} C_VEL
LIN {X 0,Y 381.927,Z 466.642,A -85,B 0,C 180,E1 17759.639,E2 17759.639} C_VEL
LIN {X 0,Y 378.935,Z 483.014,A -85,B 0,C 180,E1 17758.012,E2 17758.012} C_VEL
LIN {X 0,Y 375.91,Z 497.821,A -85,B 0,C 180,E1 17756.2,E2 17756.2} C_VEL
LIN {X 0,Y 372.736,Z 512.102,A -85,B 0,C 180,E1 17754.062,E2 17754.062} C_VEL
LIN {X 0,Y 369.797,Z 524.763,A -85,B 0,C 180,E1 17751.74,E2 17751.74} C_VEL
LIN {X 0,Y 367.162,Z 535.915,A -85,B 0,C 180,E1 17749.238,E2 17749.238} C_VEL
LIN {X 0,Y 364.93,Z 545.592,A -85,B 0,C 180,E1 17746.554,E2 17746.554} C_VEL
LIN {X 0,Y 363.149,Z 553.776,A -85,B 0,C 180,E1 17743.696,E2 17743.696} C_VEL
LIN {X 0,Y 361.853,Z 560.421,A -85,B 0,C 180,E1 17740.668,E2 17740.668} C_VEL
LIN {X 0,Y 361.06,Z 565.25,A -85,B 0,C 180,E1 17737.637,E2 17737.637} C_VEL
LIN {X 0,Y 360.637,Z 568.41,A -85,B 0,C 180,E1 17734.611,E2 17734.611} C_VEL
LIN {X 0,Y 360.577,Z 568.816,A -85,B 0,C 180,E1 17733.99,E2 17733.99} C_VEL
LIN {X 0,Y 359.499,Z 569.611,A -85,B 0,C 180,E1 17732.773,E2 17732.773} C_VEL
LIN {X 0,Y 354.634,Z 570.66,A -85,B 0,C 180,E1 17730.383,E2 17730.383} C_VEL
LIN {X 0,Y 352.608,Z 570.729,A -85,B 0,C 180,E1 17728.876,E2 17728.876} C_VEL
LIN {X 0,Y 352.488,Z 570.671,A -85,B 0,C 180,E1 17728.423,E2 17728.423} C_VEL
LIN {X 0,Y 352.683,Z 569.016,A -85,B 0,C 180,E1 17725.12,E2 17725.12} C_VEL
LIN {X 0,Y 353.184,Z 565.619,A -85,B 0,C 180,E1 17721.862,E2 17721.862} C_VEL
LIN {X 0,Y 354.071,Z 560.67,A -85,B 0,C 180,E1 17718.763,E2 17718.763} C_VEL
LIN {X 0,Y 355.493,Z 553.879,A -85,B 0,C 180,E1 17715.669,E2 17715.669} C_VEL
LIN {X 0,Y 357.429,Z 545.549,A -85,B 0,C 180,E1 17712.75,E2 17712.75} C_VEL
LIN {X 0,Y 359.838,Z 535.716,A -85,B 0,C 180,E1 17710.014,E2 17710.014} C_VEL
LIN {X 0,Y 362.678,Z 524.322,A -85,B 0,C 180,E1 17707.452,E2 17707.452} C_VEL
LIN {X 0,Y 365.786,Z 511.523,A -85,B 0,C 180,E1 17705.104,E2 17705.104} C_VEL
LIN {X 0,Y 369.024,Z 497.562,A -85,B 0,C 180,E1 17703.009,E2 17703.009} C_VEL
LIN {X 0,Y 372.22,Z 482.609,A -85,B 0,C 180,E1 17701.172,E2 17701.172} C_VEL
LIN {X 0,Y 375.328,Z 466.17,A -85,B 0,C 180,E1 17699.535,E2 17699.535} C_VEL
LIN {X 0,Y 378.148,Z 448.856,A -85,B 0,C 180,E1 17698.163,E2 17698.163} C_VEL
LIN {X 0,Y 380.528,Z 430.764,A -85,B 0,C 180,E1 17697.049,E2 17697.049} C_VEL
LIN {X 0,Y 382.391,Z 411.818,A -85,B 0,C 180,E1 17696.188,E2 17696.188} C_VEL
LIN {X 0,Y 383.64,Z 392.55,A -85,B 0,C 180,E1 17695.598,E2 17695.598} C_VEL
LIN {X 0,Y 388.811,Z 215.158,A -85,B 0,C 180,E1 17692.355,E2 17692.355} C_VEL
LIN {X 0,Y 385.212,Z 192.721,A -85,B 0,C 180,E1 17691.378,E2 17691.378} C_VEL
LIN {X 0,Y 374.772,Z 174.204,A -85,B 0,C 180,E1 17689.496,E2 17689.496} C_VEL
LIN {X 0,Y 373.584,Z 171.916,A -85,B 0,C 180,E1 17689.228,E2 17689.228} C_VEL
LIN {X 0,Y 367.762,Z 156.578,A -85,B 0,C 180,E1 17686.094,E2 17686.094} C_VEL
LIN {X 0,Y 361.452,Z 141.85,A -85,B 0,C 180,E1 17682.667,E2 17682.667} C_VEL
LIN {X 0,Y 360.254,Z 141.017,A -85,B 0,C 180,E1 17682.303,E2 17682.303} C_VEL
LIN {X 0,Y 360.172,Z 141.139,A -85,B 0,C 180,E1 17682.207,E2 17682.207} C_VEL
LIN {X 0,Y 368.431,Z 162.788,A -85,B 0,C 180,E1 17679.089,E2 17679.089} C_VEL
LIN {X 0,Y 374.413,Z 180.595,A -85,B 0,C 180,E1 17676.698,E2 17676.698} C_VEL
LIN {X 0,Y 374.07,Z 188.531,A -85,B 0,C 180,E1 17675.987,E2 17675.987} C_VEL
LIN {X 0,Y 376.738,Z 212.427,A -85,B 0,C 180,E1 17675.06,E2 17675.06} C_VEL
LIN {X 0,Y 368.545,Z 400.377,A -85,B 0,C 180,E1 17670.419,E2 17670.419} C_VEL
LIN {X 0,Y 367.479,Z 419.627,A -85,B 0,C 180,E1 17669.656,E2 17669.656} C_VEL
LIN {X 0,Y 366.102,Z 438.362,A -85,B 0,C 180,E1 17668.632,E2 17668.632} C_VEL
LIN {X 0,Y 364.478,Z 456.417,A -85,B 0,C 180,E1 17667.355,E2 17667.355} C_VEL
LIN {X 0,Y 362.607,Z 474.562,A -85,B 0,C 180,E1 17665.741,E2 17665.741} C_VEL
LIN {X 0,Y 360.76,Z 490.837,A -85,B 0,C 180,E1 17663.956,E2 17663.956} C_VEL
LIN {X 0,Y 358.92,Z 506.128,A -85,B 0,C 180,E1 17661.919,E2 17661.919} C_VEL
LIN {X 0,Y 357.177,Z 520.217,A -85,B 0,C 180,E1 17659.629,E2 17659.629} C_VEL
LIN {X 0,Y 355.671,Z 532.667,A -85,B 0,C 180,E1 17657.168,E2 17657.168} C_VEL
LIN {X 0,Y 354.451,Z 543.53,A -85,B 0,C 180,E1 17654.54,E2 17654.54} C_VEL
LIN {X 0,Y 353.58,Z 552.288,A -85,B 0,C 180,E1 17651.914,E2 17651.914} C_VEL
LIN {X 0,Y 352.983,Z 559.604,A -85,B 0,C 180,E1 17649.127,E2 17649.127} C_VEL
LIN {X 0,Y 352.647,Z 565.089,A -85,B 0,C 180,E1 17646.349,E2 17646.349} C_VEL
LIN {X 0,Y 352.505,Z 568.881,A -85,B 0,C 180,E1 17643.578,E2 17643.578} C_VEL
LIN {X 0,Y 352.503,Z 571.074,A -85,B 0,C 180,E1 17640.813,E2 17640.813} C_VEL
LIN {X 0,Y 352.595,Z 571.711,A -85,B 0,C 180,E1 17638.05,E2 17638.05} C_VEL
LIN {X 0,Y 352.83,Z 570.794,A -85,B 0,C 180,E1 17635.286,E2 17635.286} C_VEL
LIN {X 0,Y 353.27,Z 568.317,A -85,B 0,C 180,E1 17632.52,E2 17632.52} C_VEL
LIN {X 0,Y 353.973,Z 564.203,A -85,B 0,C 180,E1 17629.75,E2 17629.75} C_VEL
LIN {X 0,Y 355.039,Z 558.388,A -85,B 0,C 180,E1 17626.98,E2 17626.98} C_VEL
LIN {X 0,Y 356.528,Z 550.644,A -85,B 0,C 180,E1 17624.215,E2 17624.215} C_VEL
LIN {X 0,Y 358.365,Z 541.421,A -85,B 0,C 180,E1 17621.623,E2 17621.623} C_VEL
LIN {X 0,Y 360.637,Z 529.885,A -85,B 0,C 180,E1 17619.044,E2 17619.044} C_VEL
LIN {X 0,Y 363.002,Z 517.548,A -85,B 0,C 180,E1 17616.804,E2 17616.804} C_VEL
LIN {X 0,Y 365.647,Z 503.225,A -85,B 0,C 180,E1 17614.663,E2 17614.663} C_VEL
LIN {X 0,Y 368.535,Z 486.44,A -85,B 0,C 180,E1 17612.622,E2 17612.622} C_VEL
LIN {X 0,Y 371.095,Z 469.742,A -85,B 0,C 180,E1 17610.989,E2 17610.989} C_VEL
LIN {X 0,Y 373.585,Z 451.6,A -85,B 0,C 180,E1 17609.55,E2 17609.55} C_VEL
LIN {X 0,Y 375.923,Z 431.899,A -85,B 0,C 180,E1 17608.321,E2 17608.321} C_VEL
LIN {X 0,Y 377.868,Z 411.53,A -85,B 0,C 180,E1 17607.37,E2 17607.37} C_VEL
LIN {X 0,Y 383.157,Z 357.967,A -85,B 0,C 180,E1 17605.572,E2 17605.572} C_VEL
LIN {X 0,Y 392.534,Z 285.723,A -85,B 0,C 180,E1 17603.123,E2 17603.123} C_VEL
LIN {X 0,Y 402.888,Z 220.245,A -85,B 0,C 180,E1 17600.878,E2 17600.878} C_VEL
LIN {X 0,Y 403.865,Z 208.582,A -85,B 0,C 180,E1 17599.84,E2 17599.84} C_VEL
LIN {X 0,Y 405.436,Z 201.759,A -85,B 0,C 180,E1 17599.099,E2 17599.099} C_VEL
LIN {X 0,Y 405.565,Z 197.108,A -85,B 0,C 180,E1 17597.698,E2 17597.698} C_VEL
LIN {X 0,Y 405.889,Z 194.196,A -85,B 0,C 180,E1 17596.314,E2 17596.314} C_VEL
LIN {X 0,Y 404.041,Z 199.934,A -85,B 0,C 180,E1 17594.853,E2 17594.853} C_VEL
LIN {X 0,Y 403.7,Z 201.235,A -85,B 0,C 180,E1 17594.601,E2 17594.601} C_VEL
LIN {X 0,Y 402.331,Z 206.032,A -85,B 0,C 180,E1 17594.294,E2 17594.294} C_VEL
LIN {X 0,Y 397.673,Z 222.942,A -85,B 0,C 180,E1 17593.619,E2 17593.619} C_VEL
LIN {X 0,Y 392.149,Z 249.95,A -85,B 0,C 180,E1 17592.693,E2 17592.693} C_VEL
LIN {X 0,Y 388.393,Z 270.781,A -85,B 0,C 180,E1 17591.942,E2 17591.942} C_VEL
LIN {X 0,Y 382.523,Z 417.735,A -85,B 0,C 180,E1 17588.916,E2 17588.916} C_VEL
LIN {X 0,Y 380.667,Z 439.455,A -85,B 0,C 180,E1 17588.215,E2 17588.215} C_VEL
LIN {X 0,Y 378.253,Z 460.28,A -85,B 0,C 180,E1 17587.253,E2 17587.253} C_VEL
LIN {X 0,Y 375.486,Z 479.897,A -85,B 0,C 180,E1 17586.051,E2 17586.051} C_VEL
LIN {X 0,Y 372.433,Z 498.676,A -85,B 0,C 180,E1 17584.598,E2 17584.598} C_VEL
LIN {X 0,Y 369.224,Z 516.67,A -85,B 0,C 180,E1 17582.886,E2 17582.886} C_VEL
LIN {X 0,Y 365.973,Z 533.822,A -85,B 0,C 180,E1 17580.907,E2 17580.907} C_VEL
LIN {X 0,Y 362.703,Z 550.577,A -85,B 0,C 180,E1 17578.574,E2 17578.574} C_VEL
LIN {X 0,Y 359.771,Z 565.679,A -85,B 0,C 180,E1 17576.048,E2 17576.048} C_VEL
LIN {X 0,Y 357.303,Z 579.001,A -85,B 0,C 180,E1 17573.386,E2 17573.386} C_VEL
LIN {X 0,Y 355.343,Z 590.718,A -85,B 0,C 180,E1 17570.594,E2 17570.594} C_VEL
LIN {X 0,Y 353.841,Z 601.123,A -85,B 0,C 180,E1 17567.6,E2 17567.6} C_VEL
LIN {X 0,Y 352.845,Z 609.994,A -85,B 0,C 180,E1 17564.441,E2 17564.441} C_VEL
LIN {X 0,Y 352.338,Z 616.952,A -85,B 0,C 180,E1 17561.293,E2 17561.293} C_VEL
LIN {X 0,Y 352.174,Z 622.148,A -85,B 0,C 180,E1 17558.162,E2 17558.162} C_VEL
LIN {X 0,Y 352.188,Z 625.673,A -85,B 0,C 180,E1 17555.05,E2 17555.05} C_VEL
LIN {X 0,Y 352.247,Z 627.466,A -85,B 0,C 180,E1 17552.116,E2 17552.116} C_VEL
LIN {X 0,Y 352.269,Z 627.765,A -85,B 0,C 180,E1 17549.188,E2 17549.188} C_VEL
LIN {X 0,Y 352.216,Z 626.666,A -85,B 0,C 180,E1 17546.257,E2 17546.257} C_VEL
LIN {X 0,Y 352.171,Z 624.023,A -85,B 0,C 180,E1 17543.316,E2 17543.316} C_VEL
LIN {X 0,Y 352.23,Z 619.623,A -85,B 0,C 180,E1 17540.195,E2 17540.195} C_VEL
LIN {X 0,Y 352.55,Z 613.507,A -85,B 0,C 180,E1 17537.054,E2 17537.054} C_VEL
LIN {X 0,Y 353.251,Z 606.045,A -85,B 0,C 180,E1 17534.066,E2 17534.066} C_VEL
LIN {X 0,Y 354.531,Z 596.047,A -85,B 0,C 180,E1 17530.869,E2 17530.869} C_VEL
LIN {X 0,Y 356.408,Z 584.173,A -85,B 0,C 180,E1 17527.785,E2 17527.785} C_VEL
LIN {X 0,Y 358.818,Z 570.737,A -85,B 0,C 180,E1 17524.907,E2 17524.907} C_VEL
LIN {X 0,Y 361.587,Z 556.226,A -85,B 0,C 180,E1 17522.32,E2 17522.32} C_VEL
LIN {X 0,Y 364.554,Z 541.069,A -85,B 0,C 180,E1 17520.056,E2 17520.056} C_VEL
LIN {X 0,Y 367.719,Z 524.516,A -85,B 0,C 180,E1 17517.981,E2 17517.981} C_VEL
LIN {X 0,Y 371.123,Z 506.088,A -85,B 0,C 180,E1 17516.077,E2 17516.077} C_VEL
LIN {X 0,Y 374.304,Z 487.095,A -85,B 0,C 180,E1 17514.481,E2 17514.481} C_VEL
LIN {X 0,Y 377.21,Z 467.651,A -85,B 0,C 180,E1 17513.178,E2 17513.178} C_VEL
LIN {X 0,Y 379.709,Z 447.967,A -85,B 0,C 180,E1 17512.156,E2 17512.156} C_VEL
LIN {X 0,Y 381.743,Z 427.476,A -85,B 0,C 180,E1 17511.373,E2 17511.373} C_VEL
LIN {X 0,Y 383.091,Z 405.535,A -85,B 0,C 180,E1 17510.811,E2 17510.811} C_VEL
LIN {X 0,Y 391.065,Z 201.309,A -85,B 0,C 180,E1 17506.668,E2 17506.668} C_VEL
LIN {X 0,Y 390.356,Z 196.4,A -85,B 0,C 180,E1 17506.458,E2 17506.458} C_VEL
LIN {X 0,Y 378.917,Z 175.895,A -85,B 0,C 180,E1 17504.42,E2 17504.42} C_VEL
LIN {X 0,Y 372.519,Z 165.364,A -85,B 0,C 180,E1 17503.191,E2 17503.191} C_VEL
LIN {X 0,Y 365.922,Z 150.426,A -85,B 0,C 180,E1 17500.154,E2 17500.154} C_VEL
LIN {X 0,Y 360.253,Z 138.484,A -85,B 0,C 180,E1 17497.432,E2 17497.432} C_VEL
LIN {X 0,Y 355.724,Z 129.674,A -85,B 0,C 180,E1 17495.184,E2 17495.184} C_VEL
LIN {X 0,Y 354.14,Z 126.774,A -85,B 0,C 180,E1 17494.379,E2 17494.379} C_VEL
LIN {X 0,Y 353.85,Z 125.394,A -85,B 0,C 180,E1 17494.019,E2 17494.019} C_VEL
LIN {X 0,Y 353.835,Z 125.396,A -85,B 0,C 180,E1 17489.824,E2 17489.824} C_VEL
LIN {X 0,Y 353.832,Z 125.407,A -85,B 0,C 180,E1 17485.796,E2 17485.796} C_VEL
LIN {X 0,Y 353.822,Z 125.413,A -85,B 0,C 180,E1 17481.613,E2 17481.613} C_VEL
LIN {X 0,Y 353.813,Z 125.394,A -85,B 0,C 180,E1 17477.43,E2 17477.43} C_VEL
LIN {X 0,Y 353.809,Z 125.38,A -85,B 0,C 180,E1 17473.232,E2 17473.232} C_VEL
LIN {X 0,Y 353.814,Z 125.402,A -85,B 0,C 180,E1 17469.105,E2 17469.105} C_VEL
LIN {X 0,Y 353.818,Z 125.406,A -85,B 0,C 180,E1 17465.025,E2 17465.025} C_VEL
LIN {X 0,Y 353.825,Z 125.376,A -85,B 0,C 180,E1 17460.809,E2 17460.809} C_VEL
LIN {X 0,Y 353.83,Z 125.402,A -85,B 0,C 180,E1 17456.76,E2 17456.76} C_VEL
LIN {X 0,Y 353.853,Z 125.398,A -85,B 0,C 180,E1 17452.531,E2 17452.531} C_VEL
LIN {X 0,Y 353.829,Z 125.377,A -85,B 0,C 180,E1 17448.26,E2 17448.26} C_VEL
LIN {X 0,Y 353.83,Z 125.401,A -85,B 0,C 180,E1 17444.259,E2 17444.259} C_VEL
LIN {X 0,Y 353.823,Z 125.406,A -85,B 0,C 180,E1 17440.177,E2 17440.177} C_VEL
LIN {X 0,Y 353.816,Z 125.383,A -85,B 0,C 180,E1 17436.164,E2 17436.164} C_VEL
LIN {X 0,Y 353.808,Z 125.384,A -85,B 0,C 180,E1 17432.023,E2 17432.023} C_VEL
LIN {X 0,Y 353.803,Z 125.396,A -85,B 0,C 180,E1 17427.907,E2 17427.907} C_VEL
LIN {X 0,Y 353.799,Z 125.401,A -85,B 0,C 180,E1 17423.649,E2 17423.649} C_VEL
LIN {X 0,Y 353.83,Z 125.627,A -85,B 0,C 180,E1 17421.561,E2 17421.561} C_VEL
LIN {X 0,Y 355.13,Z 128.861,A -85,B 0,C 180,E1 17420.692,E2 17420.692} C_VEL
LIN {X 0,Y 356.085,Z 130.537,A -85,B 0,C 180,E1 17420.192,E2 17420.192} C_VEL
LIN {X 0,Y 360.562,Z 140.239,A -85,B 0,C 180,E1 17417.634,E2 17417.634} C_VEL
LIN {X 0,Y 365.669,Z 151.801,A -85,B 0,C 180,E1 17414.865,E2 17414.865} C_VEL
LIN {X 0,Y 371.233,Z 165.615,A -85,B 0,C 180,E1 17411.907,E2 17411.907} C_VEL
LIN {X 0,Y 373.892,Z 172.735,A -85,B 0,C 180,E1 17410.552,E2 17410.552} C_VEL
LIN {X 0,Y 383.897,Z 190.473,A -85,B 0,C 180,E1 17408.735,E2 17408.735} C_VEL
LIN {X 0,Y 385.486,Z 193.728,A -85,B 0,C 180,E1 17408.449,E2 17408.449} C_VEL
LIN {X 0,Y 388.824,Z 216.98,A -85,B 0,C 180,E1 17407.493,E2 17407.493} C_VEL
LIN {X 0,Y 383.514,Z 394.168,A -85,B 0,C 180,E1 17404.262,E2 17404.262} C_VEL
LIN {X 0,Y 382.189,Z 413.566,A -85,B 0,C 180,E1 17403.644,E2 17403.644} C_VEL
LIN {X 0,Y 380.345,Z 431.921,A -85,B 0,C 180,E1 17402.787,E2 17402.787} C_VEL
LIN {X 0,Y 377.968,Z 449.739,A -85,B 0,C 180,E1 17401.674,E2 17401.674} C_VEL
LIN {X 0,Y 375.062,Z 467.388,A -85,B 0,C 180,E1 17400.253,E2 17400.253} C_VEL
LIN {X 0,Y 371.918,Z 483.831,A -85,B 0,C 180,E1 17398.588,E2 17398.588} C_VEL
LIN {X 0,Y 368.761,Z 498.593,A -85,B 0,C 180,E1 17396.748,E2 17396.748} C_VEL
LIN {X 0,Y 365.444,Z 512.833,A -85,B 0,C 180,E1 17394.573,E2 17394.573} C_VEL
LIN {X 0,Y 362.365,Z 525.469,A -85,B 0,C 180,E1 17392.21,E2 17392.21} C_VEL
LIN {X 0,Y 359.596,Z 536.603,A -85,B 0,C 180,E1 17389.659,E2 17389.659} C_VEL
LIN {X 0,Y 357.242,Z 546.266,A -85,B 0,C 180,E1 17386.921,E2 17386.921} C_VEL
LIN {X 0,Y 355.357,Z 554.44,A -85,B 0,C 180,E1 17384.002,E2 17384.002} C_VEL
LIN {X 0,Y 353.979,Z 561.078,A -85,B 0,C 180,E1 17380.908,E2 17380.908} C_VEL
LIN {X 0,Y 353.131,Z 565.9,A -85,B 0,C 180,E1 17377.81,E2 17377.81} C_VEL
LIN {X 0,Y 352.677,Z 569.057,A -85,B 0,C 180,E1 17374.715,E2 17374.715} C_VEL
LIN {X 0,Y 352.486,Z 570.673,A -85,B 0,C 180,E1 17371.462,E2 17371.462} C_VEL
LIN {X 0,Y 352.488,Z 570.671,A -85,B 0,C 180,E1 17368.423,E2 17368.423} C_VEL
LIN {X 0,Y 351.567,Z 570.423,A -85,B 0,C 180,E1 17367.17,E2 17367.17} C_VEL
LIN {X 0,Y 347.465,Z 569.464,A -85,B 0,C 180,E1 17364.979,E2 17364.979} C_VEL
LIN {X 0,Y 345.216,Z 568.189,A -85,B 0,C 180,E1 17363.365,E2 17363.365} C_VEL
LIN {X 0,Y 345.047,Z 567.492,A -85,B 0,C 180,E1 17362.726,E2 17362.726} C_VEL
LIN {X 0,Y 345.849,Z 563.031,A -85,B 0,C 180,E1 17359.505,E2 17359.505} C_VEL
LIN {X 0,Y 347.169,Z 556.851,A -85,B 0,C 180,E1 17356.339,E2 17356.339} C_VEL
LIN {X 0,Y 349.016,Z 549.176,A -85,B 0,C 180,E1 17353.352,E2 17353.352} C_VEL
LIN {X 0,Y 351.335,Z 540.067,A -85,B 0,C 180,E1 17350.55,E2 17350.55} C_VEL
LIN {X 0,Y 354.09,Z 529.56,A -85,B 0,C 180,E1 17347.94,E2 17347.94} C_VEL
LIN {X 0,Y 357.176,Z 517.656,A -85,B 0,C 180,E1 17345.524,E2 17345.524} C_VEL
LIN {X 0,Y 360.495,Z 504.289,A -85,B 0,C 180,E1 17343.299,E2 17343.299} C_VEL
LIN {X 0,Y 363.83,Z 489.955,A -85,B 0,C 180,E1 17341.343,E2 17341.343} C_VEL
LIN {X 0,Y 367.024,Z 474.767,A -85,B 0,C 180,E1 17339.645,E2 17339.645} C_VEL
LIN {X 0,Y 370.134,Z 457.836,A -85,B 0,C 180,E1 17338.121,E2 17338.121} C_VEL
LIN {X 0,Y 372.746,Z 440.932,A -85,B 0,C 180,E1 17336.915,E2 17336.915} C_VEL
LIN {X 0,Y 375.029,Z 422.046,A -85,B 0,C 180,E1 17335.888,E2 17335.888} C_VEL
